KUKA KRL program: MyProgram_243().src

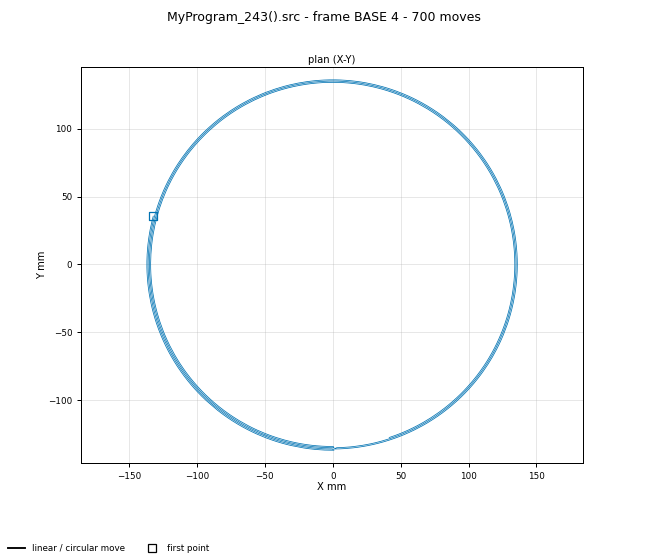
[picture p0: tool path of MyProgram_243().src in frame BASE 4, 700 of 700 moves have a stored position in this frame; points joined in program order, loops and branches not executed]
&ACCESS RVP
&REL 1
&PARAM TEMPLATE = C:\KRC\Roboter\Template\vorgabe
&PARAM EDITMASK = *
DEF MyProgram_243()
; ---- Setting reference (Base) ----
$BASE = BASE_DATA[4]

; --------------------------
; ---- Setting tool (TCP) ----
$TOOL = TOOL_DATA[3]
; --------------------------

$VEL.CP = VEL_APROX_PRINT
Startdeposition()
$VEL.CP = VEL_PRINT
LIN {X -132.1479,Y 35.5316,Z 162,A 162.612,B 22.5411,C -1.0275,E1 22.4083,E2 284.7882} C_DIS
LIN {X -132.9584,Y 32.3675,Z 162,A 163.9986,B 22.5412,C -1.024,E1 22.4074,E2 283.4017} C_DIS
LIN {X -133.7341,Y 28.9953,Z 162,A 165.3572,B 22.5416,C -1.0153,E1 22.4065,E2 282.0568} C_DIS
LIN {X -134.3965,Y 25.7509,Z 162,A 166.8499,B 22.5416,C -1.0157,E1 22.4057,E2 280.5534} C_DIS
LIN {X -134.985,Y 22.4628,Z 162,A 168.2719,B 22.5417,C -1.0122,E1 22.4051,E2 279.1309} C_DIS
LIN {X -135.5638,Y 18.6678,Z 162,A 170.017,B 22.5417,C -1.0132,E1 22.4044,E2 277.3716} C_DIS
LIN {X -136.0422,Y 14.7684,Z 162,A 171.5514,B 22.5421,C -1.0029,E1 22.4039,E2 275.8538} C_DIS
LIN {X -136.3695,Y 11.3551,Z 162,A 173.0277,B 22.5422,C -1.0001,E1 22.4035,E2 274.375} C_DIS
LIN {X -136.6388,Y 7.4678,Z 162,A 174.7811,B 22.5422,C -1.0003,E1 22.4032,E2 272.6092} C_DIS
LIN {X -136.821,Y 2.3704,Z 162,A 176.8126,B 22.5427,C -0.9887,E1 22.403,E2 270.5945} C_DIS
LIN {X -136.8263,Y -2.0499,Z 162,A 178.6813,B 22.5429,C -0.9835,E1 22.403,E2 268.7266} C_DIS
LIN {X -136.7134,Y -5.9516,Z 162,A -179.5726,B 22.5429,C -0.9833,E1 22.4033,E2 266.9694} C_DIS
LIN {X -136.4577,Y -10.2442,Z 162,A -177.8134,B 22.5432,C -0.9757,E1 22.4036,E2 265.2183} C_DIS
LIN {X -136.0949,Y -14.2787,Z 162,A -176.2336,B 22.5437,C -0.965,E1 22.404,E2 263.656} C_DIS
LIN {X -135.6787,Y -17.8001,Z 162,A -174.6843,B 22.5437,C -0.9632,E1 22.4045,E2 262.1009} C_DIS
LIN {X -135.101,Y -21.7679,Z 162,A -172.859,B 22.5437,C -0.9645,E1 22.4053,E2 260.2601} C_DIS
LIN {X -134.448,Y -25.4817,Z 162,A -171.4171,B 22.5442,C -0.9533,E1 22.406,E2 258.8378} C_DIS
LIN {X -133.8444,Y -28.4841,Z 162,A -170.0113,B 22.5441,C -0.9549,E1 22.4069,E2 257.4185} C_DIS
LIN {X -133.0086,Y -32.1595,Z 162,A -168.5445,B 22.5445,C -0.945,E1 22.4078,E2 255.9682} C_DIS
LIN {X -132.1539,Y -35.5092,Z 162,A -166.498,B 22.5436,C -0.9678,E1 22.4093,E2 253.8483} C_DIS
LIN {X -130.8595,Y -40.0158,Z 162,A -165.0549,B 22.5448,C -0.9381,E1 22.4104,E2 252.474} C_DIS
LIN {X -129.8351,Y -43.2241,Z 162,A -163.6072,B 22.5448,C -0.9356,E1 22.4117,E2 251.0236} C_DIS
LIN {X -128.378,Y -47.3813,Z 162,A -161.5655,B 22.5448,C -0.939,E1 22.4136,E2 248.9597} C_DIS
LIN {X -126.4379,Y -52.3363,Z 162,A -159.5206,B 22.5453,C -0.9242,E1 22.4157,E2 246.9411} C_DIS
LIN {X -125.0704,Y -55.5246,Z 162,A -157.4706,B 22.5444,C -0.9474,E1 22.4182,E2 244.8173} C_DIS
LIN {X -122.9248,Y -60.126,Z 162,A -155.4739,B 22.5449,C -0.9355,E1 22.4206,E2 242.8399} C_DIS
LIN {X -120.9842,Y -63.9405,Z 162,A -154.3142,B 22.5462,C -0.9014,E1 22.422,E2 241.7626} C_DIS
LIN {X -118.9843,Y -67.5927,Z 162,A -152.2799,B 22.5458,C -0.91,E1 22.4248,E2 239.6938} C_DIS
LIN {X -116.5755,Y -71.6669,Z 162,A -150.3113,B 22.5461,C -0.9041,E1 22.4276,E2 237.7294} C_DIS
LIN {X -114.3025,Y -75.2391,Z 162,A -148.0549,B 22.5454,C -0.9219,E1 22.4312,E2 235.4136} C_DIS
LIN {X -111.6085,Y -79.1811,Z 162,A -146.4975,B 22.5464,C -0.8963,E1 22.4336,E2 233.9147} C_DIS
LIN {X -109.6366,Y -81.8891,Z 162,A -145.0699,B 22.5464,C -0.894,E1 22.4359,E2 232.4854} C_DIS
LIN {X -106.8318,Y -85.5165,Z 162,A -143.1704,B 22.5467,C -0.8884,E1 22.4392,E2 230.5905} C_DIS
LIN {X -104.4579,Y -88.4003,Z 162,A -141.3214,B 22.5463,C -0.898,E1 22.4426,E2 228.7069} C_DIS
LIN {X -102.0287,Y -91.1928,Z 162,A -140.3003,B 22.5473,C -0.8699,E1 22.4444,E2 227.7543} C_DIS
LIN {X -99.6826,Y -93.7518,Z 162,A -138.5586,B 22.547,C -0.88,E1 22.4477,E2 225.9775} C_DIS
LIN {X -96.344,Y -97.1794,Z 162,A -136.6172,B 22.5472,C -0.8728,E1 22.4515,E2 224.0457} C_DIS
LIN {X -93.0775,Y -100.3126,Z 162,A -134.6531,B 22.5472,C -0.8721,E1 22.4555,E2 222.0744} C_DIS
LIN {X -84.7797,Y -107.4174,Z 162,A -130.3287,B 22.548,C -0.8514,E1 22.4647,E2 217.7853} C_DIS
LIN {X -80.9765,Y -110.3122,Z 162,A -128.1214,B 22.5478,C -0.8575,E1 22.4697,E2 215.5533} C_DIS
LIN {X -77.7183,Y -112.632,Z 162,A -126.346,B 22.5478,C -0.8594,E1 22.4737,E2 213.766} C_DIS
LIN {X -73.8799,Y -115.1857,Z 162,A -124.4429,B 22.5478,C -0.8551,E1 22.4782,E2 211.8674} C_DIS
LIN {X -69.9948,Y -117.587,Z 162,A -122.5683,B 22.5481,C -0.8504,E1 22.4826,E2 209.9985} C_DIS
LIN {X -66.2461,Y -119.739,Z 162,A -120.7348,B 22.5481,C -0.849,E1 22.4871,E2 208.1627} C_DIS
LIN {X -62.7854,Y -121.5897,Z 162,A -119.0231,B 22.5481,C -0.8501,E1 22.4914,E2 206.4428} C_DIS
LIN {X -59.1797,Y -123.3825,Z 162,A -117.3145,B 22.5481,C -0.8491,E1 22.4957,E2 204.7317} C_DIS
LIN {X -55.5104,Y -125.0767,Z 162,A -115.3139,B 22.5476,C -0.862,E1 22.5009,E2 202.692} C_DIS
LIN {X -51.6723,Y -126.7112,Z 162,A -113.931,B 22.5483,C -0.8427,E1 22.5043,E2 201.3562} C_DIS
LIN {X -48.8745,Y -127.8175,Z 162,A -112.5832,B 22.5483,C -0.8457,E1 22.5079,E2 199.9973} C_DIS
LIN {X -44.8525,Y -129.2816,Z 162,A -110.9547,B 22.5486,C -0.8362,E1 22.5121,E2 198.3899} C_DIS
LIN {X -41.5447,Y -130.3822,Z 162,A -109.4829,B 22.5486,C -0.8356,E1 22.516,E2 196.9167} C_DIS
LIN {X -37.9958,Y -131.4611,Z 162,A -107.8588,B 22.5485,C -0.838,E1 22.5204,E2 195.2835} C_DIS
LIN {X -33.7722,Y -132.6083,Z 162,A -106.1156,B 22.5487,C -0.8325,E1 22.525,E2 193.5517} C_DIS
LIN {X -30.5556,Y -133.3862,Z 162,A -104.7545,B 22.5487,C -0.8306,E1 22.5287,E2 192.1935} C_DIS
LIN {X -21.194,Y -135.1903,Z 162,A -100.7042,B 22.5487,C -0.8317,E1 22.5399,E2 188.1354} C_DIS
LIN {X -17.7477,Y -135.6855,Z 162,A -98.5879,B 22.5476,C -0.8638,E1 22.546,E2 185.9337} C_DIS
LIN {X -12.3536,Y -136.2845,Z 162,A -96.7009,B 22.5483,C -0.8445,E1 22.5511,E2 184.096} C_DIS
LIN {X -9.1175,Y -136.5392,Z 162,A -95.3192,B 22.5483,C -0.8456,E1 22.5549,E2 182.7108} C_DIS
LIN {X -5.827,Y -136.7182,Z 162,A -94.3815,B 22.549,C -0.8239,E1 22.5574,E2 181.8294} C_DIS
LIN {X 0.956,Y -136.8378,Z 162,A -91.1377,B 22.5483,C -0.8443,E1 22.5666,E2 178.5323} C_DIS
Enddeposition()
LIN {X 0.956,Y -136.8378,Z 162,A -91.1377,B 22.5483,C -0.8443,E1 22.5666,E2 178.5323} C_DIS
Startdeposition()
$VEL.CP = VEL_PRINT
LIN {X -0.2334,Y -135.9196,Z 162,A -92.5282,B 21.3065,C -0.6019,E1 21.3126,E2 180.4426} C_DIS
LIN {X -3.8269,Y -135.8649,Z 162,A -93.5596,B 21.3059,C -0.6237,E1 21.3099,E2 181.4142} C_DIS
LIN {X -7.1029,Y -135.7333,Z 162,A -95.1398,B 21.3062,C -0.6146,E1 21.3054,E2 183.0199} C_DIS
LIN {X -13.5908,Y -135.2388,Z 162,A -98.0002,B 21.3063,C -0.6094,E1 21.2974,E2 185.896} C_DIS
LIN {X -17.7059,Y -134.7604,Z 162,A -99.5578,B 21.3061,C -0.6183,E1 21.2932,E2 187.4305} C_DIS
LIN {X -21.7349,Y -134.171,Z 162,A -101.4303,B 21.3062,C -0.6118,E1 21.2879,E2 189.3229} C_DIS
LIN {X -28.2019,Y -132.9613,Z 162,A -103.9064,B 21.3058,C -0.6262,E1 21.2813,E2 191.7624} C_DIS
LIN {X -32.3871,Y -132.0045,Z 162,A -105.8123,B 21.3059,C -0.6229,E1 21.276,E2 193.6806} C_DIS
LIN {X -35.1696,Y -131.2895,Z 162,A -107.0688,B 21.3059,C -0.6216,E1 21.2726,E2 194.9428} C_DIS
LIN {X -38.4295,Y -130.3727,Z 162,A -108.5181,B 21.3059,C -0.6216,E1 21.2687,E2 196.3948} C_DIS
LIN {X -42.4293,Y -129.1272,Z 162,A -110.4038,B 21.3061,C -0.6177,E1 21.2637,E2 198.2954} C_DIS
LIN {X -46.4957,Y -127.7188,Z 162,A -112.3466,B 21.3061,C -0.6136,E1 21.2585,E2 200.2541} C_DIS
LIN {X -55.1136,Y -124.2434,Z 162,A -116.0722,B 21.3058,C -0.6261,E1 21.249,E2 203.9553} C_DIS
LIN {X -58.8057,Y -122.5386,Z 162,A -117.7449,B 21.3058,C -0.6299,E1 21.2448,E2 205.6224} C_DIS
LIN {X -62.2944,Y -120.8042,Z 162,A -119.3789,B 21.3057,C -0.6324,E1 21.2407,E2 207.2549} C_DIS
LIN {X -65.536,Y -119.0775,Z 162,A -121.0522,B 21.3057,C -0.629,E1 21.2365,E2 208.9432} C_DIS
LIN {X -69.4336,Y -116.8473,Z 162,A -122.9199,B 21.3057,C -0.6328,E1 21.232,E2 210.807} C_DIS
LIN {X -73.1219,Y -114.5753,Z 162,A -124.7704,B 21.3057,C -0.6345,E1 21.2277,E2 212.6598} C_DIS
LIN {X -76.9602,Y -112.0331,Z 162,A -126.6969,B 21.3055,C -0.6383,E1 21.2232,E2 214.5835} C_DIS
LIN {X -80.6257,Y -109.4249,Z 162,A -128.6706,B 21.3055,C -0.6382,E1 21.2187,E2 216.5658} C_DIS
LIN {X -83.2917,Y -107.4094,Z 162,A -130.0276,B 21.3054,C -0.6429,E1 21.2157,E2 217.9155} C_DIS
LIN {X -86.9347,Y -104.4832,Z 162,A -132.4983,B 21.3059,C -0.6251,E1 21.2103,E2 220.4466} C_DIS
LIN {X -90.5729,Y -101.3452,Z 162,A -134.0516,B 21.3052,C -0.6493,E1 21.2072,E2 221.9404} C_DIS
LIN {X -93.8703,Y -98.2987,Z 162,A -135.85,B 21.305,C -0.6572,E1 21.2035,E2 223.7257} C_DIS
LIN {X -96.946,Y -95.2668,Z 162,A -137.5121,B 21.3046,C -0.6679,E1 21.2003,E2 225.3667} C_DIS
LIN {X -99.0485,Y -93.0793,Z 162,A -139.0778,B 21.3049,C -0.6584,E1 21.1972,E2 226.9669} C_DIS
LIN {X -102.0742,Y -89.7511,Z 162,A -141.0897,B 21.3049,C -0.6577,E1 21.1934,E2 228.9914} C_DIS
LIN {X -105.3855,Y -85.8384,Z 162,A -143.1221,B 21.3046,C -0.6682,E1 21.1898,E2 231.0058} C_DIS
LIN {X -108.1096,Y -82.3812,Z 162,A -144.9286,B 21.3044,C -0.6748,E1 21.1867,E2 232.8045} C_DIS
LIN {X -110.4942,Y -79.1539,Z 162,A -146.6977,B 21.3044,C -0.6756,E1 21.1838,E2 234.5814} C_DIS
LIN {X -113.3531,Y -75.0031,Z 162,A -148.6448,B 21.304,C -0.6885,E1 21.1808,E2 236.5044} C_DIS
LIN {X -115.2076,Y -72.1223,Z 162,A -150.3202,B 21.3042,C -0.6825,E1 21.1783,E2 238.2067} C_DIS
LIN {X -117.4639,Y -68.3859,Z 162,A -152.1255,B 21.304,C -0.6888,E1 21.1757,E2 240.0056} C_DIS
LIN {X -119.6677,Y -64.4511,Z 162,A -154.0117,B 21.3038,C -0.6946,E1 21.1732,E2 241.8877} C_DIS
LIN {X -121.1916,Y -61.5335,Z 162,A -155.3534,B 21.3036,C -0.7004,E1 21.1714,E2 243.2219} C_DIS
LIN {X -124.3228,Y -54.9361,Z 162,A -158.4447,B 21.3034,C -0.7085,E1 21.1678,E2 246.311} C_DIS
LIN {X -125.5052,Y -52.1752,Z 162,A -159.7449,B 21.3034,C -0.7107,E1 21.1664,E2 247.6137} C_DIS
LIN {X -126.8199,Y -48.894,Z 162,A -161.2631,B 21.3032,C -0.7138,E1 21.1648,E2 249.1334} C_DIS
LIN {X -128.294,Y -44.8841,Z 162,A -163.1444,B 21.3032,C -0.7158,E1 21.163,E2 251.0221} C_DIS
LIN {X -129.5273,Y -41.1886,Z 162,A -164.7044,B 21.3029,C -0.7241,E1 21.1617,E2 252.5696} C_DIS
LIN {X -130.563,Y -37.7794,Z 162,A -166.5203,B 21.3032,C -0.7155,E1 21.1602,E2 254.4219} C_DIS
LIN {X -131.434,Y -34.6278,Z 162,A -167.5885,B 21.3026,C -0.7326,E1 21.1595,E2 255.4501} C_DIS
LIN {X -132.3079,Y -31.1286,Z 162,A -169.276,B 21.3026,C -0.7303,E1 21.1584,E2 257.1559} C_DIS
LIN {X -133.2279,Y -26.9106,Z 162,A -170.9656,B 21.3023,C -0.7413,E1 21.1574,E2 258.8268} C_DIS
LIN {X -133.7716,Y -24.0628,Z 162,A -172.2202,B 21.3023,C -0.7438,E1 21.1568,E2 260.0835} C_DIS
LIN {X -134.3449,Y -20.6232,Z 162,A -173.671,B 21.3021,C -0.7492,E1 21.1561,E2 261.5297} C_DIS
LIN {X -134.8662,Y -16.8982,Z 162,A -175.2631,B 21.3019,C -0.7538,E1 21.1556,E2 263.1203} C_DIS
LIN {X -135.1826,Y -14.132,Z 162,A -176.5632,B 21.3019,C -0.7523,E1 21.1552,E2 264.4339} C_DIS
LIN {X -135.5553,Y -9.9317,Z 162,A -178.2889,B 21.3017,C -0.7601,E1 21.1548,E2 266.1503} C_DIS
LIN {X -135.793,Y -5.8728,Z 162,A 179.9148,B 21.3017,C -0.7621,E1 21.1545,E2 267.9541} C_DIS
LIN {X -135.9038,Y -2.0291,Z 162,A 178.401,B 21.3013,C -0.7717,E1 21.1545,E2 269.4521} C_DIS
LIN {X -135.901,Y 2.1995,Z 162,A 176.5657,B 21.3012,C -0.7752,E1 21.1545,E2 271.2909} C_DIS
LIN {X -135.7975,Y 5.7565,Z 162,A 175.1116,B 21.3009,C -0.7819,E1 21.1545,E2 272.7369} C_DIS
LIN {X -135.6057,Y 9.2415,Z 162,A 173.5075,B 21.3009,C -0.7811,E1 21.1549,E2 274.3548} C_DIS
LIN {X -135.2923,Y 13.033,Z 162,A 171.9109,B 21.3008,C -0.7866,E1 21.1553,E2 275.9478} C_DIS
LIN {X -134.7943,Y 17.4468,Z 162,A 170.0685,B 21.3005,C -0.7938,E1 21.1559,E2 277.7834} C_DIS
LIN {X -134.3075,Y 20.8651,Z 162,A 168.6193,B 21.3003,C -0.7987,E1 21.1565,E2 279.2293} C_DIS
LIN {X -133.7052,Y 24.4337,Z 162,A 167.0858,B 21.3002,C -0.8032,E1 21.1572,E2 280.7613} C_DIS
LIN {X -132.9189,Y 28.3983,Z 162,A 165.3214,B 21.3001,C -0.8061,E1 21.1582,E2 282.5301} C_DIS
LIN {X -132.1192,Y 31.9113,Z 162,A 163.8484,B 21.2998,C -0.8127,E1 21.1591,E2 283.995} C_DIS
LIN {X -131.2604,Y 35.2787,Z 162,A 162.3572,B 21.2998,C -0.8162,E1 21.1602,E2 285.4869} C_DIS
LIN {X -130.2348,Y 38.9002,Z 162,A 160.7651,B 21.2995,C -0.8209,E1 21.1614,E2 287.077} C_DIS
LIN {X -129.1239,Y 42.4391,Z 162,A 159.126,B 21.2995,C -0.8226,E1 21.1628,E2 288.7226} C_DIS
LIN {X -127.8789,Y 46.0518,Z 162,A 157.5218,B 21.2993,C -0.8279,E1 21.1643,E2 290.3232} C_DIS
LIN {X -126.4348,Y 49.8846,Z 162,A 155.8123,B 21.2991,C -0.8338,E1 21.166,E2 292.0278} C_DIS
LIN {X -124.6618,Y 54.1596,Z 162,A 153.8509,B 21.2989,C -0.8392,E1 21.1681,E2 293.9871} C_DIS
LIN {X -123.2442,Y 57.3124,Z 162,A 152.347,B 21.2988,C -0.8416,E1 21.1699,E2 295.4942} C_DIS
LIN {X -121.3485,Y 61.2251,Z 162,A 150.6714,B 21.2983,C -0.8536,E1 21.1719,E2 297.1476} C_DIS
LIN {X -118.0764,Y 67.322,Z 162,A 147.6014,B 21.2983,C -0.8555,E1 21.176,E2 300.2315} C_DIS
LIN {X -116.2087,Y 70.4973,Z 162,A 145.9945,B 21.2982,C -0.8577,E1 21.1783,E2 301.8424} C_DIS
LIN {X -114.0464,Y 73.9439,Z 162,A 144.2065,B 21.2981,C -0.8594,E1 21.181,E2 303.6364} C_DIS
LIN {X -110.7896,Y 78.7407,Z 162,A 141.8266,B 21.2977,C -0.8687,E1 21.1848,E2 306.0046} C_DIS
LIN {X -106.8612,Y 83.9939,Z 162,A 139.0312,B 21.2975,C -0.8748,E1 21.1895,E2 308.7992} C_DIS
LIN {X -102.9226,Y 88.7763,Z 162,A 136.4415,B 21.2972,C -0.8823,E1 21.1941,E2 311.3822} C_DIS
LIN {X -100.3087,Y 91.7201,Z 162,A 134.6734,B 21.2972,C -0.8819,E1 21.1974,E2 313.1609} C_DIS
LIN {X -97.2658,Y 94.9407,Z 162,A 132.7521,B 21.2972,C -0.8842,E1 21.2012,E2 315.0859} C_DIS
LIN {X -94.0928,Y 98.0861,Z 162,A 130.8858,B 21.2969,C -0.8893,E1 21.2049,E2 316.9473} C_DIS
LIN {X -90.9182,Y 101.0359,Z 162,A 129.0267,B 21.2969,C -0.8921,E1 21.2087,E2 318.8076} C_DIS
LIN {X -87.6094,Y 103.9181,Z 162,A 127.2544,B 21.2965,C -0.8994,E1 21.2124,E2 320.5679} C_DIS
LIN {X -84.4386,Y 106.5104,Z 162,A 125.3203,B 21.2967,C -0.8943,E1 21.2167,E2 322.5247} C_DIS
LIN {X -80.6388,Y 109.4153,Z 162,A 123.3832,B 21.2964,C -0.9018,E1 21.221,E2 324.4495} C_DIS
LIN {X -75.1849,Y 113.2326,Z 162,A 120.4463,B 21.2964,C -0.9017,E1 21.2278,E2 327.3985} C_DIS
LIN {X -70.65,Y 116.1163,Z 162,A 118.3043,B 21.296,C -0.9111,E1 21.2328,E2 329.5226} C_DIS
LIN {X -66.7886,Y 118.3792,Z 162,A 116.2717,B 21.2962,C -0.9081,E1 21.2378,E2 331.5706} C_DIS
LIN {X -61.6496,Y 121.1324,Z 162,A 113.9949,B 21.2957,C -0.9199,E1 21.2434,E2 333.8224} C_DIS
LIN {X -58.3357,Y 122.7631,Z 162,A 112.49,B 21.2955,C -0.9245,E1 21.2471,E2 335.3192} C_DIS
LIN {X -54.6496,Y 124.4499,Z 162,A 110.8257,B 21.2953,C -0.9289,E1 21.2513,E2 336.9762} C_DIS
LIN {X -52.2373,Y 125.4793,Z 162,A 109.3523,B 21.2959,C -0.9146,E1 21.2553,E2 338.493} C_DIS
LIN {X -48.9956,Y 126.7804,Z 162,A 108.2083,B 21.2952,C -0.9306,E1 21.2581,E2 339.5956} C_DIS
LIN {X -45.4252,Y 128.1048,Z 162,A 106.6215,B 21.2952,C -0.9334,E1 21.2623,E2 341.1786} C_DIS
LIN {X -42.5094,Y 129.1005,Z 162,A 105.3219,B 21.2951,C -0.9349,E1 21.2657,E2 342.477} C_DIS
LIN {X -35.9614,Y 131.0764,Z 162,A 102.4892,B 21.2948,C -0.9401,E1 21.2733,E2 345.3009} C_DIS
LIN {X -31.8419,Y 132.1359,Z 162,A 100.5975,B 21.2949,C -0.9375,E1 21.2784,E2 347.2031} C_DIS
LIN {X -28.6415,Y 132.8664,Z 162,A 99.2454,B 21.2949,C -0.9401,E1 21.2821,E2 348.5501} C_DIS
LIN {X -25.4806,Y 133.5087,Z 162,A 97.8355,B 21.2949,C -0.9389,E1 21.286,E2 349.965} C_DIS
LIN {X -22.2396,Y 134.0868,Z 162,A 96.4615,B 21.2949,C -0.9405,E1 21.2897,E2 351.3363} C_DIS
LIN {X -18.9892,Y 134.5857,Z 162,A 95.0405,B 21.2949,C -0.9398,E1 21.2937,E2 352.7606} C_DIS
LIN {X -13.679,Y 135.2303,Z 162,A 92.7643,B 21.2949,C -0.94,E1 21.3,E2 355.0379} C_DIS
LIN {X -9.9539,Y 135.5537,Z 162,A 91.1718,B 21.2949,C -0.94,E1 21.3044,E2 356.6313} C_DIS
LIN {X -6.3293,Y 135.7721,Z 162,A 89.7311,B 21.2947,C -0.9445,E1 21.3084,E2 358.0602} C_DIS
LIN {X -2.3794,Y 135.898,Z 162,A 87.9675,B 21.2948,C -0.9405,E1 21.3134,E2 359.8348} C_DIS
LIN {X 2.0503,Y 135.9034,Z 162,A 86.1664,B 21.2947,C -0.9437,E1 21.3184,E2 361.6269} C_DIS
LIN {X 5.7146,Y 135.7992,Z 162,A 84.657,B 21.2947,C -0.9454,E1 21.3226,E2 363.1313} C_DIS
LIN {X 10.3482,Y 135.5249,Z 162,A 82.6398,B 21.2947,C -0.9426,E1 21.3282,E2 365.1551} C_DIS
LIN {X 13.4186,Y 135.2553,Z 162,A 81.287,B 21.2948,C -0.94,E1 21.332,E2 366.514} C_DIS
LIN {X 17.5932,Y 134.7751,Z 162,A 79.5677,B 21.2948,C -0.942,E1 21.3367,E2 368.2264} C_DIS
LIN {X 20.864,Y 134.3076,Z 162,A 77.8795,B 21.2953,C -0.9283,E1 21.3415,E2 369.9504} C_DIS
LIN {X 24.3503,Y 133.7201,Z 162,A 76.7633,B 21.2947,C -0.9445,E1 21.3444,E2 371.0206} C_DIS
LIN {X 27.8278,Y 133.0413,Z 162,A 75.2567,B 21.2947,C -0.9432,E1 21.3486,E2 372.5286} C_DIS
LIN {X 30.5921,Y 132.4313,Z 162,A 74.0865,B 21.2947,C -0.9436,E1 21.3517,E2 373.6958} C_DIS
LIN {X 33.5926,Y 131.7018,Z 162,A 72.7585,B 21.2947,C -0.9416,E1 21.3554,E2 375.0269} C_DIS
LIN {X 36.7603,Y 130.853,Z 162,A 71.3771,B 21.2948,C -0.9407,E1 21.3591,E2 376.4081} C_DIS
LIN {X 39.9209,Y 129.9236,Z 162,A 69.916,B 21.295,C -0.9363,E1 21.363,E2 377.8781} C_DIS
LIN {X 43.3175,Y 128.8314,Z 162,A 68.1588,B 21.2955,C -0.9235,E1 21.3677,E2 379.6664} C_DIS
LIN {X 46.5345,Y 127.7049,Z 162,A 66.244,B 21.2965,C -0.9005,E1 21.3729,E2 381.6395} C_DIS
LIN {X 52.0712,Y 125.5486,Z 162,A 64.7367,B 21.2947,C -0.9433,E1 21.3765,E2 383.0252} C_DIS
LIN {X 55.7247,Y 123.97,Z 162,A 62.8499,B 21.2952,C -0.9318,E1 21.3814,E2 384.9382} C_DIS
LIN {X 59.0495,Y 122.422,Z 162,A 61.3314,B 21.2952,C -0.9312,E1 21.3852,E2 386.4537} C_DIS
LIN {X 61.9759,Y 120.9663,Z 162,A 59.9154,B 21.2954,C -0.9276,E1 21.3888,E2 387.8748} C_DIS
LIN {X 65.6585,Y 119.0097,Z 162,A 58.0907,B 21.2956,C -0.9221,E1 21.3933,E2 389.7083} C_DIS
LIN {X 69.5194,Y 116.7962,Z 162,A 56.2584,B 21.2956,C -0.9214,E1 21.3977,E2 391.536} C_DIS
LIN {X 73.2636,Y 114.4846,Z 162,A 54.3926,B 21.2958,C -0.918,E1 21.4021,E2 393.404} C_DIS
LIN {X 77.0918,Y 111.9428,Z 162,A 52.4689,B 21.2958,C -0.9154,E1 21.4065,E2 395.3271} C_DIS
LIN {X 81.2712,Y 108.9463,Z 162,A 50.5979,B 21.2954,C -0.9255,E1 21.4107,E2 397.1625} C_DIS
LIN {X 88.4978,Y 103.1625,Z 162,A 46.7313,B 21.2957,C -0.9197,E1 21.4192,E2 401.0275} C_DIS
LIN {X 91.8269,Y 100.2105,Z 162,A 44.5748,B 21.2964,C -0.9027,E1 21.4237,E2 403.2202} C_DIS
LIN {X 94.9661,Y 97.2409,Z 162,A 42.9591,B 21.2961,C -0.9086,E1 21.4269,E2 404.8118} C_DIS
LIN {X 97.176,Y 95.0323,Z 162,A 41.4452,B 21.2966,C -0.8965,E1 21.4299,E2 406.3512} C_DIS
LIN {X 100.1432,Y 91.9002,Z 162,A 39.5007,B 21.297,C -0.8865,E1 21.4336,E2 408.3129} C_DIS
LIN {X 103.4604,Y 88.1491,Z 162,A 37.5101,B 21.297,C -0.8874,E1 21.4373,E2 410.2904} C_DIS
LIN {X 106.4331,Y 84.5358,Z 162,A 35.4801,B 21.2973,C -0.8799,E1 21.4408,E2 412.3296} C_DIS
LIN {X 108.7196,Y 81.5749,Z 162,A 33.3572,B 21.2984,C -0.8503,E1 21.4445,E2 414.5214} C_DIS
LIN {X 111.9869,Y 77.0275,Z 162,A 31.9068,B 21.297,C -0.8874,E1 21.4467,E2 415.8617} C_DIS
LIN {X 113.7639,Y 74.379,Z 162,A 30.2771,B 21.2977,C -0.8703,E1 21.4492,E2 417.5285} C_DIS
LIN {X 116.1563,Y 70.5839,Z 162,A 28.4077,B 21.2978,C -0.8664,E1 21.452,E2 419.3973} C_DIS
LIN {X 118.3523,Y 66.8363,Z 162,A 26.5908,B 21.298,C -0.8622,E1 21.4545,E2 421.2146} C_DIS
LIN {X 120.461,Y 62.9519,Z 162,A 24.8895,B 21.2979,C -0.8649,E1 21.4567,E2 422.8978} C_DIS
LIN {X 122.1881,Y 59.5336,Z 162,A 23.2546,B 21.2981,C -0.8594,E1 21.4588,E2 424.5374} C_DIS
LIN {X 123.4847,Y 56.7923,Z 162,A 21.9888,B 21.2982,C -0.8564,E1 21.4603,E2 425.8032} C_DIS
LIN {X 124.8021,Y 53.8349,Z 162,A 20.5998,B 21.2984,C -0.8513,E1 21.4618,E2 427.197} C_DIS
LIN {X 126.3015,Y 50.2205,Z 162,A 18.7033,B 21.299,C -0.8346,E1 21.4638,E2 429.1266} C_DIS
LIN {X 129.0338,Y 42.7098,Z 162,A 15.0167,B 21.3,C -0.8095,E1 21.4672,E2 432.8571} C_DIS
LIN {X 130.5435,Y 37.846,Z 162,A 13.5687,B 21.299,C -0.8366,E1 21.4683,E2 434.2212} C_DIS
LIN {X 131.3307,Y 35.015,Z 162,A 12.2659,B 21.2992,C -0.8297,E1 21.4693,E2 435.5339} C_DIS
LIN {X 132.1821,Y 31.6503,Z 162,A 10.8073,B 21.2994,C -0.8255,E1 21.4703,E2 436.9941} C_DIS
LIN {X 132.9609,Y 28.2037,Z 162,A 9.4265,B 21.2994,C -0.8261,E1 21.4711,E2 438.3635} C_DIS
LIN {X 133.5085,Y 25.4818,Z 162,A 8.165,B 21.2996,C -0.8181,E1 21.4718,E2 439.6381} C_DIS
LIN {X 134.2214,Y 21.4212,Z 162,A 6.2718,B 21.3001,C -0.8051,E1 21.4727,E2 441.5535} C_DIS
LIN {X 134.8708,Y 16.8617,Z 162,A 4.4116,B 21.3001,C -0.8029,E1 21.4733,E2 443.4066} C_DIS
LIN {X 135.3133,Y 12.8141,Z 162,A 2.7455,B 21.3003,C -0.8,E1 21.4738,E2 445.069} C_DIS
LIN {X 135.6885,Y 7.919,Z 162,A 0.677,B 21.3005,C -0.7934,E1 21.4742,E2 447.1407} C_DIS
LIN {X 135.8661,Y 3.7808,Z 162,A -0.9786,B 21.3005,C -0.7923,E1 21.4744,E2 448.7878} C_DIS
LIN {X 135.9212,Y -0.1669,Z 162,A -2.79,B 21.301,C -0.7798,E1 21.4744,E2 450.6205} C_DIS
LIN {X 135.8354,Y -4.7856,Z 162,A -4.5729,B 21.301,C -0.7815,E1 21.4743,E2 452.3859} C_DIS
LIN {X 135.6696,Y -8.2265,Z 162,A -5.988,B 21.301,C -0.7787,E1 21.4741,E2 453.7987} C_DIS
LIN {X 135.3816,Y -12.0885,Z 162,A -7.6074,B 21.3012,C -0.7741,E1 21.4737,E2 455.4193} C_DIS
LIN {X 135.0135,Y -15.6655,Z 162,A -9.3366,B 21.3017,C -0.7589,E1 21.4731,E2 457.1778} C_DIS
LIN {X 134.2632,Y -21.151,Z 162,A -11.4057,B 21.3015,C -0.7643,E1 21.4723,E2 459.2176} C_DIS
LIN {X 133.7707,Y -24.0677,Z 162,A -12.6976,B 21.3018,C -0.7581,E1 21.4717,E2 460.5172} C_DIS
LIN {X 133.0162,Y -27.9478,Z 162,A -14.4194,B 21.302,C -0.7501,E1 21.4707,E2 462.2489} C_DIS
LIN {X 131.8917,Y -32.8445,Z 162,A -16.3162,B 21.3019,C -0.7542,E1 21.4695,E2 464.1215} C_DIS
LIN {X 130.7338,Y -37.1864,Z 162,A -18.2734,B 21.3022,C -0.7452,E1 21.4681,E2 466.0898} C_DIS
LIN {X 129.6235,Y -40.8873,Z 162,A -20.2572,B 21.3029,C -0.7229,E1 21.4664,E2 468.121} C_DIS
LIN {X 128.5078,Y -44.2674,Z 162,A -21.1751,B 21.3021,C -0.7466,E1 21.4657,E2 468.9682} C_DIS
LIN {X 125.7263,Y -51.6457,Z 162,A -24.7839,B 21.3029,C -0.7224,E1 21.462,E2 472.6189} C_DIS
LIN {X 124.0015,Y -55.6545,Z 162,A -26.5262,B 21.3029,C -0.7217,E1 21.4601,E2 474.352} C_DIS
LIN {X 122.4879,Y -58.9117,Z 162,A -28.0176,B 21.3031,C -0.7183,E1 21.4583,E2 475.8431} C_DIS
LIN {X 120.6786,Y -62.5377,Z 162,A -29.8002,B 21.3033,C -0.7096,E1 21.456,E2 477.6381} C_DIS
LIN {X 117.5764,Y -68.1916,Z 162,A -32.284,B 21.3033,C -0.7131,E1 21.4527,E2 480.0968} C_DIS
LIN {X 114.3258,Y -73.5118,Z 162,A -35.0612,B 21.3037,C -0.6984,E1 21.4486,E2 482.8973} C_DIS
LIN {X 110.9812,Y -78.4697,Z 162,A -37.4222,B 21.3037,C -0.6992,E1 21.4449,E2 485.2422} C_DIS
LIN {X 108.885,Y -81.3535,Z 162,A -39.1174,B 21.3041,C -0.6859,E1 21.442,E2 486.9642} C_DIS
LIN {X 106.1867,Y -84.8453,Z 162,A -40.9316,B 21.3041,C -0.6832,E1 21.4389,E2 488.7756} C_DIS
LIN {X 103.4742,Y -88.1328,Z 162,A -42.7384,B 21.3043,C -0.6781,E1 21.4357,E2 490.5865} C_DIS
LIN {X 100.4722,Y -91.5407,Z 162,A -44.6313,B 21.3044,C -0.6743,E1 21.4321,E2 492.4797} C_DIS
LIN {X 97.5178,Y -94.6816,Z 162,A -46.4227,B 21.3045,C -0.6711,E1 21.4287,E2 494.2705} C_DIS
LIN {X 94.7258,Y -97.4749,Z 162,A -48.1433,B 21.3047,C -0.6645,E1 21.4253,E2 496.0007} C_DIS
LIN {X 91.3653,Y -100.6314,Z 162,A -50.0386,B 21.3048,C -0.6623,E1 21.4214,E2 497.8927} C_DIS
LIN {X 88.052,Y -103.5429,Z 162,A -51.8966,B 21.3049,C -0.6582,E1 21.4174,E2 499.7533} C_DIS
LIN {X 84.5904,Y -106.3896,Z 162,A -53.7678,B 21.305,C -0.6549,E1 21.4134,E2 501.625} C_DIS
LIN {X 80.9725,Y -109.1687,Z 162,A -55.6773,B 21.3051,C -0.6516,E1 21.4091,E2 503.5354} C_DIS
LIN {X 77.3228,Y -111.7837,Z 162,A -57.5893,B 21.3053,C -0.6468,E1 21.4048,E2 505.4524} C_DIS
LIN {X 73.6704,Y -114.224,Z 162,A -59.4343,B 21.3053,C -0.6436,E1 21.4004,E2 507.299} C_DIS
LIN {X 69.6042,Y -116.7456,Z 162,A -61.3715,B 21.3053,C -0.6436,E1 21.3958,E2 509.2288} C_DIS
LIN {X 65.7737,Y -118.9458,Z 162,A -63.4378,B 21.3057,C -0.6308,E1 21.3907,E2 511.323} C_DIS
LIN {X 60.0343,Y -121.9411,Z 162,A -65.9312,B 21.3055,C -0.6375,E1 21.3846,E2 513.79} C_DIS
LIN {X 56.4086,Y -123.6621,Z 162,A -67.7346,B 21.3057,C -0.6296,E1 21.38,E2 515.6094} C_DIS
LIN {X 51.8056,Y -125.6596,Z 162,A -69.7892,B 21.3057,C -0.6294,E1 21.3747,E2 517.6587} C_DIS
LIN {X 47.9137,Y -127.1932,Z 162,A -71.8054,B 21.3061,C -0.6153,E1 21.3694,E2 519.7085} C_DIS
LIN {X 44.5649,Y -128.4046,Z 162,A -72.9651,B 21.3058,C -0.6293,E1 21.3664,E2 520.8269} C_DIS
LIN {X 41.1726,Y -129.5324,Z 162,A -74.5035,B 21.3058,C -0.6261,E1 21.3623,E2 522.3707} C_DIS
LIN {X 36.936,Y -130.8039,Z 162,A -76.4062,B 21.306,C -0.6223,E1 21.3572,E2 524.2799} C_DIS
LIN {X 33.2447,Y -131.7901,Z 162,A -77.9143,B 21.3059,C -0.6254,E1 21.3532,E2 525.7766} C_DIS
LIN {X 30.0368,Y -132.5582,Z 162,A -79.2964,B 21.3059,C -0.6245,E1 21.3494,E2 527.1588} C_DIS
LIN {X 26.509,Y -133.3097,Z 162,A -80.8135,B 21.3059,C -0.6234,E1 21.3453,E2 528.6768} C_DIS
LIN {X 22.7358,Y -134.004,Z 162,A -82.4793,B 21.306,C -0.6199,E1 21.3407,E2 530.3499} C_DIS
LIN {X 18.458,Y -134.6614,Z 162,A -84.2298,B 21.306,C -0.6221,E1 21.3359,E2 532.0925} C_DIS
LIN {X 15.0722,Y -135.0814,Z 162,A -85.8831,B 21.3063,C -0.6114,E1 21.3312,E2 533.7739} C_DIS
LIN {X 9.132,Y -135.6137,Z 162,A -88.3368,B 21.3063,C -0.613,E1 21.3244,E2 536.2216} C_DIS
LIN {X 5.1747,Y -135.8202,Z 162,A -89.921,B 21.3061,C -0.6164,E1 21.32,E2 537.7959} C_DIS
LIN {X 0.9468,Y -135.9079,Z 162,A -91.1941,B 21.3055,C -0.6394,E1 21.3166,E2 539.0054} C_DIS
Enddeposition()
LIN {X 0.9468,Y -135.9079,Z 162,A -91.1941,B 21.3055,C -0.6394,E1 21.3166,E2 539.0054} C_DIS
Startdeposition()
$VEL.CP = VEL_PRINT
LIN {X 2.9964,Y -134.9648,Z 162,A -89.8352,B 20.1418,C -0.4915,E1 20.1525,E2 537.9529} C_DIS
LIN {X 6.3819,Y -134.8456,Z 162,A -88.3556,B 20.1418,C -0.4938,E1 20.1566,E2 536.4671} C_DIS
LIN {X 9.7799,Y -134.6412,Z 162,A -87.0405,B 20.1419,C -0.4888,E1 20.1603,E2 535.1674} C_DIS
LIN {X 12.4989,Y -134.4166,Z 162,A -85.931,B 20.1419,C -0.4872,E1 20.1633,E2 534.0633} C_DIS
LIN {X 15.216,Y -134.1378,Z 162,A -84.5171,B 20.1417,C -0.4989,E1 20.1673,E2 532.6166} C_DIS
LIN {X 18.6912,Y -133.6962,Z 162,A -83.1451,B 20.1417,C -0.4948,E1 20.1711,E2 531.258} C_DIS
LIN {X 21.907,Y -133.2067,Z 162,A -81.7452,B 20.1417,C -0.4966,E1 20.175,E2 529.8547} C_DIS
LIN {X 24.9399,Y -132.6726,Z 162,A -80.6014,B 20.1419,C -0.4904,E1 20.1781,E2 528.7303} C_DIS
LIN {X 27.7029,Y -132.1251,Z 162,A -79.1445,B 20.1416,C -0.5029,E1 20.1821,E2 527.2397} C_DIS
LIN {X 31.3327,Y -131.3095,Z 162,A -77.6527,B 20.1416,C -0.5005,E1 20.1862,E2 525.7575} C_DIS
LIN {X 35.5712,Y -130.2274,Z 162,A -75.7102,B 20.1415,C -0.5061,E1 20.1914,E2 523.8026} C_DIS
LIN {X 39.0964,Y -129.2109,Z 162,A -74.4231,B 20.1417,C -0.4958,E1 20.1948,E2 522.548} C_DIS
LIN {X 41.8652,Y -128.3425,Z 162,A -72.9154,B 20.1414,C -0.5095,E1 20.1989,E2 521.0044} C_DIS
LIN {X 45.0037,Y -127.2759,Z 162,A -71.5195,B 20.1414,C -0.5107,E1 20.2026,E2 519.6085} C_DIS
LIN {X 48.5056,Y -125.9809,Z 162,A -70.0594,B 20.1414,C -0.5072,E1 20.2064,E2 518.1624} C_DIS
LIN {X 51.6195,Y -124.7373,Z 162,A -68.6395,B 20.1414,C -0.5091,E1 20.21,E2 516.7414} C_DIS
LIN {X 54.7168,Y -123.41,Z 162,A -67.2204,B 20.1414,C -0.5106,E1 20.2137,E2 515.3222} C_DIS
LIN {X 57.4276,Y -122.1743,Z 162,A -65.8291,B 20.1412,C -0.5182,E1 20.2172,E2 513.9135} C_DIS
LIN {X 60.4848,Y -120.69,Z 162,A -64.5146,B 20.1412,C -0.5147,E1 20.2205,E2 512.6136} C_DIS
LIN {X 63.6963,Y -119.0258,Z 162,A -62.8729,B 20.1412,C -0.522,E1 20.2246,E2 510.9566} C_DIS
LIN {X 67.8288,Y -116.7202,Z 162,A -60.9061,B 20.1411,C -0.5236,E1 20.2294,E2 508.9926} C_DIS
LIN {X 71.5152,Y -114.4986,Z 162,A -59.0864,B 20.141,C -0.5266,E1 20.2337,E2 507.1715} C_DIS
LIN {X 74.7667,Y -112.4023,Z 162,A -57.5289,B 20.141,C -0.5259,E1 20.2373,E2 505.6226} C_DIS
LIN {X 78.0881,Y -110.1211,Z 162,A -55.7417,B 20.1408,C -0.5328,E1 20.2414,E2 503.8235} C_DIS
LIN {X 81.666,Y -107.4949,Z 162,A -53.9518,B 20.1408,C -0.5324,E1 20.2454,E2 502.0428} C_DIS
LIN {X 84.5732,Y -105.2223,Z 162,A -52.3936,B 20.1408,C -0.5353,E1 20.2488,E2 500.4836} C_DIS
LIN {X 87.609,Y -102.7084,Z 162,A -50.6513,B 20.1406,C -0.5421,E1 20.2526,E2 498.7302} C_DIS
LIN {X 90.9781,Y -99.7367,Z 162,A -48.7458,B 20.1405,C -0.5464,E1 20.2565,E2 496.822} C_DIS
LIN {X 94.2145,Y -96.6856,Z 162,A -46.957,B 20.1405,C -0.5462,E1 20.2601,E2 495.0431} C_DIS
LIN {X 96.6856,Y -94.2145,Z 162,A -45.4077,B 20.1403,C -0.5528,E1 20.2632,E2 493.4833} C_DIS
LIN {X 99.6826,Y -91.0377,Z 162,A -43.5616,B 20.1403,C -0.557,E1 20.2667,E2 491.6353} C_DIS
LIN {X 102.5732,Y -87.768,Z 162,A -41.8007,B 20.1402,C -0.5574,E1 20.2699,E2 489.8832} C_DIS
LIN {X 104.8062,Y -85.089,Z 162,A -40.2785,B 20.14,C -0.5631,E1 20.2726,E2 488.3534} C_DIS
LIN {X 107.4264,Y -81.7556,Z 162,A -38.4918,B 20.14,C -0.5673,E1 20.2757,E2 486.5656} C_DIS
LIN {X 109.7412,Y -78.6204,Z 162,A -36.8113,B 20.1398,C -0.5729,E1 20.2784,E2 484.8791} C_DIS
LIN {X 112.0368,Y -75.3142,Z 162,A -35.2061,B 20.1398,C -0.5728,E1 20.2809,E2 483.2844} C_DIS
LIN {X 114.0392,Y -72.2455,Z 162,A -33.6629,B 20.1397,C -0.5765,E1 20.2833,E2 481.7401} C_DIS
LIN {X 116.1234,Y -68.8459,Z 162,A -31.9712,B 20.1395,C -0.5812,E1 20.2857,E2 480.0458} C_DIS
LIN {X 117.9923,Y -65.5909,Z 162,A -30.2923,B 20.1393,C -0.5897,E1 20.288,E2 478.3534} C_DIS
LIN {X 120.1017,Y -61.6404,Z 162,A -28.634,B 20.1395,C -0.5841,E1 20.2902,E2 476.7227} C_DIS
LIN {X 121.6176,Y -58.5927,Z 162,A -27.086,B 20.1392,C -0.593,E1 20.2921,E2 475.1594} C_DIS
LIN {X 122.8858,Y -55.8887,Z 162,A -25.8293,B 20.1392,C -0.5962,E1 20.2936,E2 473.902} C_DIS
LIN {X 124.3602,Y -52.5224,Z 162,A -24.3953,B 20.1392,C -0.5951,E1 20.2951,E2 472.4812} C_DIS
LIN {X 125.5196,Y -49.6921,Z 162,A -22.9958,B 20.1389,C -0.6037,E1 20.2966,E2 471.0669} C_DIS
LIN {X 126.8464,Y -46.1948,Z 162,A -21.3812,B 20.1387,C -0.6097,E1 20.2982,E2 469.4462} C_DIS
LIN {X 127.9469,Y -43.0531,Z 162,A -20.0248,B 20.1387,C -0.6114,E1 20.2994,E2 468.0946} C_DIS
LIN {X 128.8446,Y -40.2932,Z 162,A -18.8018,B 20.1386,C -0.6148,E1 20.3004,E2 466.8708} C_DIS
LIN {X 129.8924,Y -36.769,Z 162,A -17.2565,B 20.1385,C -0.6189,E1 20.3016,E2 465.3248} C_DIS
LIN {X 130.743,Y -33.6196,Z 162,A -16.0294,B 20.1385,C -0.6159,E1 20.3025,E2 464.1152} C_DIS
LIN {X 131.4264,Y -30.8478,Z 162,A -14.5679,B 20.1381,C -0.6312,E1 20.3035,E2 462.6203} C_DIS
LIN {X 132.2015,Y -27.3272,Z 162,A -13.3119,B 20.1383,C -0.6234,E1 20.3042,E2 461.3963} C_DIS
LIN {X 132.7443,Y -24.5647,Z 162,A -11.9852,B 20.138,C -0.6332,E1 20.3049,E2 460.0511} C_DIS
LIN {X 133.3432,Y -21.0623,Z 162,A -10.6331,B 20.1381,C -0.6308,E1 20.3055,E2 458.7162} C_DIS
LIN {X 133.7494,Y -18.3186,Z 162,A -9.2137,B 20.1377,C -0.6457,E1 20.3061,E2 457.2643} C_DIS
LIN {X 134.1776,Y -14.8462,Z 162,A -7.9947,B 20.1379,C -0.6381,E1 20.3065,E2 456.0765} C_DIS
LIN {X 134.4791,Y -11.8097,Z 162,A -6.4867,B 20.1375,C -0.652,E1 20.3069,E2 454.5396} C_DIS
LIN {X 134.7346,Y -8.3961,Z 162,A -5.1187,B 20.1375,C -0.6527,E1 20.3071,E2 453.1799} C_DIS
LIN {X 134.878,Y -5.656,Z 162,A -3.9829,B 20.1374,C -0.655,E1 20.3073,E2 452.0459} C_DIS
LIN {X 134.9648,Y -2.9964,Z 162,A -2.864,B 20.1373,C -0.6581,E1 20.3073,E2 450.9266} C_DIS
LIN {X 134.9978,Y 0.3023,Z 162,A -1.3289,B 20.1369,C -0.6688,E1 20.3073,E2 449.3723} C_DIS
LIN {X 134.9307,Y 4.226,Z 162,A 0.3065,B 20.1369,C -0.6727,E1 20.3073,E2 447.7381} C_DIS
LIN {X 134.765,Y 7.9031,Z 162,A 1.5947,B 20.1371,C -0.6649,E1 20.3071,E2 446.4819} C_DIS
LIN {X 134.5507,Y 10.9618,Z 162,A 3.0253,B 20.1367,C -0.675,E1 20.3068,E2 445.033} C_DIS
LIN {X 134.2448,Y 14.2214,Z 162,A 4.4381,B 20.1366,C -0.6804,E1 20.3064,E2 443.6153} C_DIS
LIN {X 133.8528,Y 17.5297,Z 162,A 5.8378,B 20.1364,C -0.6841,E1 20.3059,E2 442.2153} C_DIS
LIN {X 133.3432,Y 21.0623,Z 162,A 7.4728,B 20.1361,C -0.6944,E1 20.3052,E2 440.5629} C_DIS
LIN {X 132.6726,Y 24.9399,Z 162,A 9.039,B 20.1361,C -0.6947,E1 20.3044,E2 439.0074} C_DIS
LIN {X 131.6997,Y 29.6511,Z 162,A 11.0056,B 20.1361,C -0.6975,E1 20.3033,E2 437.0473} C_DIS
LIN {X 130.9134,Y 32.9479,Z 162,A 12.4607,B 20.1358,C -0.7026,E1 20.3023,E2 435.588} C_DIS
LIN {X 130.0357,Y 36.2567,Z 162,A 13.7948,B 20.1358,C -0.7015,E1 20.3013,E2 434.2668} C_DIS
LIN {X 129.2109,Y 39.0964,Z 162,A 14.9782,B 20.1358,C -0.702,E1 20.3004,E2 433.0908} C_DIS
LIN {X 128.3425,Y 41.8652,Z 162,A 16.4701,B 20.1353,C -0.7176,E1 20.2991,E2 431.5647} C_DIS
LIN {X 127.2759,Y 45.0037,Z 162,A 17.8921,B 20.1352,C -0.7224,E1 20.2978,E2 430.1389} C_DIS
LIN {X 125.9809,Y 48.5056,Z 162,A 19.3229,B 20.1352,C -0.7199,E1 20.2964,E2 428.7253} C_DIS
LIN {X 124.7373,Y 51.6195,Z 162,A 20.7373,B 20.1352,C -0.7236,E1 20.2949,E2 427.3102} C_DIS
LIN {X 123.41,Y 54.7168,Z 162,A 22.1967,B 20.1349,C -0.729,E1 20.2933,E2 425.8453} C_DIS
LIN {X 122.1743,Y 57.4276,Z 162,A 23.5381,B 20.1347,C -0.736,E1 20.2917,E2 424.4928} C_DIS
LIN {X 120.69,Y 60.4848,Z 162,A 24.8485,B 20.1347,C -0.734,E1 20.2901,E2 423.1973} C_DIS
LIN {X 119.0258,Y 63.6963,Z 162,A 26.4858,B 20.1345,C -0.7428,E1 20.2879,E2 421.5454} C_DIS
LIN {X 116.7202,Y 67.8288,Z 162,A 28.4478,B 20.1343,C -0.7461,E1 20.2852,E2 419.587} C_DIS
LIN {X 114.4986,Y 71.5152,Z 162,A 30.2639,B 20.1342,C -0.7503,E1 20.2826,E2 417.7703} C_DIS
LIN {X 112.2632,Y 74.9752,Z 162,A 31.9845,B 20.1341,C -0.7535,E1 20.2799,E2 416.0513} C_DIS
LIN {X 110.0663,Y 78.1658,Z 162,A 33.611,B 20.134,C -0.7568,E1 20.2773,E2 414.4254} C_DIS
LIN {X 107.614,Y 81.5081,Z 162,A 35.3322,B 20.1339,C -0.7594,E1 20.2744,E2 412.7073} C_DIS
LIN {X 105.2223,Y 84.5732,Z 162,A 36.9485,B 20.1338,C -0.7618,E1 20.2716,E2 411.0937} C_DIS
LIN {X 102.7084,Y 87.609,Z 162,A 38.6903,B 20.1335,C -0.7688,E1 20.2685,E2 409.3419} C_DIS
LIN {X 99.823,Y 90.8829,Z 162,A 40.5353,B 20.1334,C -0.7726,E1 20.2651,E2 407.4961} C_DIS
LIN {X 97.1479,Y 93.737,Z 162,A 42.193,B 20.1333,C -0.7761,E1 20.2619,E2 405.8375} C_DIS
LIN {X 94.2145,Y 96.6856,Z 162,A 43.8604,B 20.1333,C -0.7755,E1 20.2586,E2 404.181} C_DIS
LIN {X 91.5198,Y 99.2394,Z 162,A 45.4256,B 20.1332,C -0.7782,E1 20.2554,E2 402.6159} C_DIS
LIN {X 88.4663,Y 101.9713,Z 162,A 47.1626,B 20.1331,C -0.7816,E1 20.2517,E2 400.878} C_DIS
LIN {X 85.6024,Y 104.3867,Z 162,A 48.7396,B 20.133,C -0.784,E1 20.2484,E2 399.3016} C_DIS
LIN {X 82.8802,Y 106.5609,Z 162,A 50.3151,B 20.1327,C -0.791,E1 20.2449,E2 397.7132} C_DIS
LIN {X 79.5748,Y 109.052,Z 162,A 51.9588,B 20.1327,C -0.7891,E1 20.2412,E2 396.0827} C_DIS
LIN {X 76.7455,Y 111.0613,Z 162,A 53.4788,B 20.1326,C -0.7937,E1 20.2377,E2 394.5561} C_DIS
LIN {X 73.3209,Y 113.3507,Z 162,A 55.2423,B 20.1325,C -0.7971,E1 20.2336,E2 392.7899} C_DIS
LIN {X 69.6633,Y 115.6347,Z 162,A 57.0638,B 20.1324,C -0.7995,E1 20.2293,E2 390.9687} C_DIS
LIN {X 65.7703,Y 117.893,Z 162,A 59.0213,B 20.1322,C -0.8044,E1 20.2245,E2 389.0048} C_DIS
LIN {X 61.6404,Y 120.1017,Z 162,A 60.7141,B 20.1326,C -0.7941,E1 20.2204,E2 387.3477} C_DIS
LIN {X 58.5927,Y 121.6176,Z 162,A 62.3059,B 20.1323,C -0.8023,E1 20.2164,E2 385.7374} C_DIS
LIN {X 55.577,Y 123.0253,Z 162,A 63.5842,B 20.1324,C -0.7981,E1 20.2132,E2 384.4755} C_DIS
LIN {X 52.4029,Y 124.4101,Z 162,A 65.0151,B 20.1324,C -0.7981,E1 20.2095,E2 383.0491} C_DIS
LIN {X 49.6921,Y 125.5196,Z 162,A 66.4158,B 20.1321,C -0.8062,E1 20.2058,E2 381.6289} C_DIS
LIN {X 46.0997,Y 126.8807,Z 162,A 67.9897,B 20.1321,C -0.8053,E1 20.2017,E2 380.0618} C_DIS
LIN {X 43.0597,Y 127.9447,Z 162,A 69.402,B 20.1321,C -0.8085,E1 20.198,E2 378.6438} C_DIS
LIN {X 40.2932,Y 128.8446,Z 162,A 70.633,B 20.132,C -0.8093,E1 20.1947,E2 377.4133} C_DIS
LIN {X 36.769,Y 129.8924,Z 162,A 72.1877,B 20.132,C -0.8103,E1 20.1905,E2 375.8594} C_DIS
LIN {X 33.4984,Y 130.7737,Z 162,A 73.6504,B 20.1319,C -0.8123,E1 20.1866,E2 374.3937} C_DIS
LIN {X 28.8986,Y 131.8669,Z 162,A 75.6216,B 20.1319,C -0.8119,E1 20.1812,E2 372.4272} C_DIS
LIN {X 26.1328,Y 132.4445,Z 162,A 76.9472,B 20.1317,C -0.8179,E1 20.1776,E2 371.0863} C_DIS
LIN {X 22.9988,Y 133.0246,Z 162,A 78.2821,B 20.1317,C -0.8176,E1 20.1739,E2 369.7538} C_DIS
LIN {X 19.8755,Y 133.5269,Z 162,A 79.5067,B 20.1319,C -0.813,E1 20.1706,E2 368.544} C_DIS
LIN {X 16.2158,Y 134.0186,Z 162,A 81.103,B 20.1318,C -0.8147,E1 20.1661,E2 366.9446} C_DIS
LIN {X 12.8421,Y 134.3837,Z 162,A 82.418,B 20.132,C -0.8096,E1 20.1625,E2 365.6454} C_DIS
LIN {X 10.228,Y 134.6085,Z 162,A 83.4793,B 20.132,C -0.8075,E1 20.1596,E2 364.5909} C_DIS
LIN {X 7.5381,Y 134.7875,Z 162,A 84.8707,B 20.1317,C -0.818,E1 20.1556,E2 363.1698} C_DIS
LIN {X 4.1434,Y 134.9329,Z 162,A 86.2379,B 20.1317,C -0.8148,E1 20.1518,E2 361.8123} C_DIS
LIN {X 0.6774,Y 134.9943,Z 162,A 87.6797,B 20.1318,C -0.8134,E1 20.1478,E2 360.3748} C_DIS
LIN {X -2.9964,Y 134.9648,Z 162,A 89.2316,B 20.1318,C -0.8128,E1 20.1435,E2 358.8247} C_DIS
LIN {X -6.3819,Y 134.8456,Z 162,A 90.6734,B 20.1318,C -0.8126,E1 20.1395,E2 357.3831} C_DIS
LIN {X -9.6282,Y 134.6523,Z 162,A 92.0737,B 20.1318,C -0.8129,E1 20.1356,E2 355.9812} C_DIS
LIN {X -12.906,Y 134.3775,Z 162,A 93.4688,B 20.1318,C -0.8123,E1 20.1317,E2 354.5871} C_DIS
LIN {X -17.137,Y 133.9043,Z 162,A 95.271,B 20.1319,C -0.8112,E1 20.1267,E2 352.7867} C_DIS
LIN {X -19.8755,Y 133.5269,Z 162,A 96.5824,B 20.1317,C -0.8162,E1 20.123,E2 351.4592} C_DIS
LIN {X -23.3735,Y 132.9575,Z 162,A 97.9573,B 20.132,C -0.8098,E1 20.1193,E2 350.1013} C_DIS
LIN {X -26.1328,Y 132.4445,Z 162,A 99.1523,B 20.132,C -0.8091,E1 20.116,E2 348.9068} C_DIS
LIN {X -29.6511,Y 131.6997,Z 162,A 100.6844,B 20.132,C -0.8081,E1 20.1118,E2 347.3752} C_DIS
LIN {X -32.8772,Y 130.9314,Z 162,A 102.109,B 20.132,C -0.8075,E1 20.108,E2 345.9496} C_DIS
LIN {X -35.5712,Y 130.2274,Z 162,A 103.404,B 20.132,C -0.811,E1 20.1044,E2 344.6419} C_DIS
LIN {X -39.0964,Y 129.2109,Z 162,A 104.6975,B 20.1324,C -0.7986,E1 20.1011,E2 343.3819} C_DIS
LIN {X -41.9303,Y 128.3208,Z 162,A 106.213,B 20.1321,C -0.8077,E1 20.097,E2 341.8366} C_DIS
LIN {X -45.0037,Y 127.2759,Z 162,A 107.6193,B 20.1321,C -0.8072,E1 20.0932,E2 340.4282} C_DIS
LIN {X -48.6449,Y 125.9267,Z 162,A 109.1107,B 20.1324,C -0.7987,E1 20.0894,E2 338.9575} C_DIS
LIN {X -51.6195,Y 124.7373,Z 162,A 110.5186,B 20.1324,C -0.7989,E1 20.0857,E2 337.5451} C_DIS
LIN {X -54.7168,Y 123.41,Z 162,A 111.9582,B 20.1324,C -0.7973,E1 20.0821,E2 336.1059} C_DIS
LIN {X -57.921,Y 121.9385,Z 162,A 113.4197,B 20.1326,C -0.7937,E1 20.0784,E2 334.6504} C_DIS
LIN {X -60.4848,Y 120.69,Z 162,A 114.6753,B 20.1326,C -0.7937,E1 20.0752,E2 333.3907} C_DIS
LIN {X -63.9576,Y 118.8853,Z 162,A 116.3957,B 20.1326,C -0.7934,E1 20.071,E2 331.665} C_DIS
LIN {X -67.8288,Y 116.7202,Z 162,A 118.3153,B 20.1326,C -0.7917,E1 20.0663,E2 329.7431} C_DIS
LIN {X -71.5152,Y 114.4986,Z 162,A 120.152,B 20.1328,C -0.7888,E1 20.0619,E2 327.9074} C_DIS
LIN {X -74.7667,Y 112.4023,Z 162,A 121.7245,B 20.133,C -0.783,E1 20.0583,E2 326.3455} C_DIS
LIN {X -77.6267,Y 110.4466,Z 162,A 123.2031,B 20.133,C -0.7805,E1 20.0549,E2 324.8678} C_DIS
LIN {X -80.8051,Y 108.1428,Z 162,A 124.9046,B 20.1332,C -0.7786,E1 20.0511,E2 323.1642} C_DIS
LIN {X -83.7295,Y 105.8955,Z 162,A 126.4529,B 20.1333,C -0.7747,E1 20.0477,E2 321.62} C_DIS
LIN {X -86.5952,Y 103.5645,Z 162,A 128.1163,B 20.1333,C -0.7752,E1 20.0441,E2 319.9472} C_DIS
LIN {X -89.7406,Y 100.8519,Z 162,A 129.9154,B 20.1333,C -0.7728,E1 20.0403,E2 318.1461} C_DIS
LIN {X -92.9552,Y 97.8969,Z 162,A 131.6676,B 20.1337,C -0.7645,E1 20.0367,E2 316.4088} C_DIS
LIN {X -95.4581,Y 95.4581,Z 162,A 133.1599,B 20.1337,C -0.7614,E1 20.0338,E2 314.9176} C_DIS
LIN {X -97.8969,Y 92.9552,Z 162,A 134.7053,B 20.1338,C -0.7604,E1 20.0308,E2 313.3668} C_DIS
LIN {X -100.7626,Y 89.8403,Z 162,A 136.5284,B 20.1339,C -0.7571,E1 20.0274,E2 311.543} C_DIS
LIN {X -103.5645,Y 86.5952,Z 162,A 138.317,B 20.1342,C -0.7513,E1 20.0241,E2 309.761} C_DIS
LIN {X -106.0242,Y 83.5656,Z 162,A 139.9576,B 20.1343,C -0.7464,E1 20.0213,E2 308.1248} C_DIS
LIN {X -108.1428,Y 80.8051,Z 162,A 141.5549,B 20.1343,C -0.7473,E1 20.0186,E2 306.5151} C_DIS
LIN {X -110.5662,Y 77.4571,Z 162,A 143.2095,B 20.1346,C -0.7387,E1 20.0159,E2 304.8755} C_DIS
LIN {X -112.5173,Y 74.5945,Z 162,A 144.7421,B 20.1346,C -0.7372,E1 20.0135,E2 303.3375} C_DIS
LIN {X -114.4986,Y 71.5152,Z 162,A 146.339,B 20.1347,C -0.7346,E1 20.0111,E2 301.7379} C_DIS
LIN {X -116.7202,Y 67.8288,Z 162,A 148.2059,B 20.1349,C -0.7311,E1 20.0085,E2 299.8689} C_DIS
LIN {X -119.0258,Y 63.6963,Z 162,A 150.2632,B 20.1349,C -0.7273,E1 20.0057,E2 297.8089} C_DIS
LIN {X -120.69,Y 60.4848,Z 162,A 151.7844,B 20.1352,C -0.7223,E1 20.0038,E2 296.2919} C_DIS
LIN {X -122.3444,Y 57.0597,Z 162,A 153.3019,B 20.1355,C -0.7138,E1 20.002,E2 294.7888} C_DIS
LIN {X -123.5752,Y 54.3476,Z 162,A 154.697,B 20.1355,C -0.7152,E1 20.0004,E2 293.3799} C_DIS
LIN {X -124.8924,Y 51.2481,Z 162,A 155.9962,B 20.1357,C -0.7059,E1 19.999,E2 292.0988} C_DIS
LIN {X -126.1259,Y 48.1324,Z 162,A 157.5501,B 20.1357,C -0.7068,E1 19.9975,E2 290.5312} C_DIS
LIN {X -127.4462,Y 44.5125,Z 162,A 159.0559,B 20.136,C -0.6968,E1 19.9961,E2 289.0438} C_DIS
LIN {X -128.4626,Y 41.489,Z 162,A 160.2866,B 20.1363,C -0.6878,E1 19.995,E2 287.8304} C_DIS
LIN {X -129.3261,Y 38.72,Z 162,A 161.7966,B 20.1361,C -0.6949,E1 19.9938,E2 286.2884} C_DIS
LIN {X -130.3279,Y 35.1943,Z 162,A 163.2954,B 20.1363,C -0.6879,E1 19.9926,E2 284.799} C_DIS
LIN {X -131.047,Y 32.4218,Z 162,A 164.4661,B 20.1365,C -0.6824,E1 19.9919,E2 283.6359} C_DIS
LIN {X -131.8669,Y 28.8986,Z 162,A 166.0106,B 20.1366,C -0.678,E1 19.9909,E2 282.0927} C_DIS
LIN {X -132.5509,Y 25.5765,Z 162,A 167.2449,B 20.137,C -0.6655,E1 19.9902,E2 280.8857} C_DIS
LIN {X -133.0246,Y 22.9988,Z 162,A 168.6959,B 20.1367,C -0.6752,E1 19.9895,E2 279.3953} C_DIS
LIN {X -133.6005,Y 19.361,Z 162,A 170.1418,B 20.137,C -0.6657,E1 19.9889,E2 277.9662} C_DIS
LIN {X -134.0117,Y 16.2729,Z 162,A 171.449,B 20.1372,C -0.661,E1 19.9885,E2 276.663} C_DIS
LIN {X -134.3041,Y 13.6708,Z 162,A 172.6027,B 20.1372,C -0.6591,E1 19.9881,E2 275.506} C_DIS
LIN {X -134.6085,Y 10.228,Z 162,A 173.9388,B 20.1376,C -0.6494,E1 19.9878,E2 274.1881} C_DIS
LIN {X -134.7954,Y 7.3795,Z 162,A 175.3595,B 20.1374,C -0.6537,E1 19.9876,E2 272.7439} C_DIS
LIN {X -134.9329,Y 4.1434,Z 162,A 176.5442,B 20.1378,C -0.6419,E1 19.9874,E2 271.5845} C_DIS
LIN {X -134.9898,Y 1.4949,Z 162,A 177.8699,B 20.1376,C -0.6462,E1 19.9874,E2 270.236} C_DIS
LIN {X -134.9838,Y -1.8542,Z 162,A 179.1101,B 20.138,C -0.6347,E1 19.9874,E2 269.0201} C_DIS
LIN {X -134.9124,Y -4.7732,Z 162,A -179.4255,B 20.1379,C -0.6396,E1 19.9875,E2 267.5301} C_DIS
LIN {X -134.7382,Y -8.3374,Z 162,A -177.9249,B 20.138,C -0.6343,E1 19.9878,E2 266.0335} C_DIS
LIN {X -134.4166,Y -12.4989,Z 162,A -176.3229,B 20.1384,C -0.6221,E1 19.9881,E2 264.4549} C_DIS
LIN {X -134.1378,Y -15.216,Z 162,A -174.895,B 20.1382,C -0.629,E1 19.9886,E2 262.9959} C_DIS
LIN {X -133.6962,Y -18.6912,Z 162,A -173.4726,B 20.1384,C -0.6219,E1 19.9891,E2 261.5837} C_DIS
LIN {X -133.2093,Y -21.8914,Z 162,A -172.1449,B 20.1386,C -0.6158,E1 19.9897,E2 260.2635} C_DIS
LIN {X -132.6726,Y -24.9399,Z 162,A -170.9412,B 20.1388,C -0.6074,E1 19.9903,E2 259.0753} C_DIS
LIN {X -132.1251,Y -27.7029,Z 162,A -169.4691,B 20.1386,C -0.6147,E1 19.9911,E2 257.5711} C_DIS
LIN {X -131.3356,Y -31.2244,Z 162,A -168.19,B 20.139,C -0.6001,E1 19.9919,E2 256.325} C_DIS
LIN {X -130.6474,Y -33.9964,Z 162,A -166.8183,B 20.139,C -0.6027,E1 19.9928,E2 254.9356} C_DIS
LIN {X -129.6767,Y -37.5225,Z 162,A -165.2517,B 20.139,C -0.5986,E1 19.994,E2 253.3691} C_DIS
LIN {X -128.8446,Y -40.2932,Z 162,A -164.0128,B 20.1392,C -0.5954,E1 19.995,E2 252.1306} C_DIS
LIN {X -127.6748,Y -43.853,Z 162,A -162.3812,B 20.1392,C -0.5924,E1 19.9965,E2 250.496} C_DIS
LIN {X -126.5713,Y -46.9435,Z 162,A -161.0028,B 20.1394,C -0.5878,E1 19.9978,E2 249.1212} C_DIS
LIN {X -125.3695,Y -50.0644,Z 162,A -159.5712,B 20.1394,C -0.5842,E1 19.9993,E2 247.6899} C_DIS
LIN {X -124.0841,Y -53.1704,Z 162,A -158.1323,B 20.1396,C -0.5806,E1 20.0008,E2 246.2513} C_DIS
LIN {X -122.8852,Y -55.8902,Z 162,A -156.8604,B 20.1396,C -0.5775,E1 20.0023,E2 244.9798} C_DIS
LIN {X -121.2624,Y -59.3243,Z 162,A -155.3904,B 20.1399,C -0.5674,E1 20.004,E2 243.529} C_DIS
LIN {X -119.9166,Y -62.0039,Z 162,A -153.8261,B 20.1397,C -0.5755,E1 20.0061,E2 241.9303} C_DIS
LIN {X -117.7924,Y -65.9492,Z 162,A -151.9222,B 20.1398,C -0.5705,E1 20.0086,E2 240.0284} C_DIS
LIN {X -115.4435,Y -69.9793,Z 162,A -150.002,B 20.14,C -0.5629,E1 20.0113,E2 238.1177} C_DIS
LIN {X -113.3507,Y -73.3209,Z 162,A -148.3552,B 20.1402,C -0.5575,E1 20.0138,E2 236.4759} C_DIS
LIN {X -111.1355,Y -76.6374,Z 162,A -146.6354,B 20.1402,C -0.5544,E1 20.0165,E2 234.7546} C_DIS
LIN {X -108.8182,Y -79.893,Z 162,A -144.8687,B 20.1403,C -0.5531,E1 20.0194,E2 232.9808} C_DIS
LIN {X -106.4333,Y -83.0448,Z 162,A -143.1372,B 20.1403,C -0.5512,E1 20.0224,E2 231.2441} C_DIS
LIN {X -103.6987,Y -86.4353,Z 162,A -141.3936,B 20.1406,C -0.5427,E1 20.0254,E2 229.5152} C_DIS
LIN {X -101.2917,Y -89.2432,Z 162,A -139.7279,B 20.1406,C -0.543,E1 20.0285,E2 227.8389} C_DIS
LIN {X -98.3529,Y -92.4719,Z 162,A -137.8428,B 20.1406,C -0.5403,E1 20.0321,E2 225.9513} C_DIS
LIN {X -95.4581,Y -95.4581,Z 162,A -136.053,B 20.1407,C -0.5375,E1 20.0356,E2 224.1599} C_DIS
LIN {X -92.3198,Y -98.4963,Z 162,A -134.2335,B 20.1408,C -0.5323,E1 20.0393,E2 222.346} C_DIS
LIN {X -89.0867,Y -101.43,Z 162,A -132.3966,B 20.141,C -0.528,E1 20.0431,E2 220.5123} C_DIS
LIN {X -85.9246,Y -104.1216,Z 162,A -130.5999,B 20.141,C -0.5261,E1 20.0469,E2 218.7124} C_DIS
LIN {X -82.5258,Y -106.8356,Z 162,A -128.7452,B 20.141,C -0.5232,E1 20.051,E2 216.8577} C_DIS
LIN {X -79.04,Y -109.4396,Z 162,A -126.9447,B 20.1412,C -0.5181,E1 20.0551,E2 215.064} C_DIS
LIN {X -75.6748,Y -111.7927,Z 162,A -125.1553,B 20.1412,C -0.5172,E1 20.0592,E2 213.2696} C_DIS
LIN {X -72.2455,Y -114.0392,Z 162,A -123.4754,B 20.1414,C -0.512,E1 20.0631,E2 211.5979} C_DIS
LIN {X -68.9248,Y -116.0764,Z 162,A -121.7911,B 20.1414,C -0.5108,E1 20.0671,E2 209.9104} C_DIS
LIN {X -65.5909,Y -117.9923,Z 162,A -120.0675,B 20.1414,C -0.5124,E1 20.0714,E2 208.1759} C_DIS
LIN {X -61.6404,Y -120.1017,Z 162,A -118.2394,B 20.1414,C -0.5069,E1 20.0759,E2 206.3573} C_DIS
LIN {X -58.5927,Y -121.6176,Z 162,A -116.8269,B 20.1415,C -0.5038,E1 20.0794,E2 204.9492} C_DIS
LIN {X -55.4268,Y -123.0924,Z 162,A -115.5331,B 20.1418,C -0.4942,E1 20.0826,E2 203.6792} C_DIS
LIN {X -52.8001,Y -124.2442,Z 162,A -114.1219,B 20.1416,C -0.501,E1 20.0863,E2 202.2442} C_DIS
LIN {X -49.2064,Y -125.7084,Z 162,A -112.4522,B 20.1416,C -0.5003,E1 20.0906,E2 200.5717} C_DIS
LIN {X -46.1948,Y -126.8464,Z 162,A -111.2549,B 20.1418,C -0.492,E1 20.0937,E2 199.3956} C_DIS
LIN {X -43.0597,Y -127.9447,Z 162,A -109.6935,B 20.1418,C -0.4971,E1 20.0979,E2 197.8154} C_DIS
LIN {X -39.879,Y -128.9714,Z 162,A -108.3204,B 20.1418,C -0.4941,E1 20.1015,E2 196.448} C_DIS
LIN {X -36.6942,Y -129.9133,Z 162,A -106.886,B 20.1418,C -0.4941,E1 20.1054,E2 195.0104} C_DIS
LIN {X -33.6196,Y -130.743,Z 162,A -105.6582,B 20.1419,C -0.4881,E1 20.1086,E2 193.798} C_DIS
LIN {X -30.8478,Y -131.4264,Z 162,A -104.1827,B 20.1417,C -0.4986,E1 20.1127,E2 192.2894} C_DIS
LIN {X -27.3272,Y -132.2015,Z 162,A -102.9151,B 20.1419,C -0.4868,E1 20.1161,E2 191.0543} C_DIS
LIN {X -24.5647,Y -132.7443,Z 162,A -101.5762,B 20.1419,C -0.4924,E1 20.1198,E2 189.6973} C_DIS
LIN {X -21.0623,Y -133.3432,Z 162,A -100.0006,B 20.1418,C -0.4948,E1 20.1242,E2 188.1128} C_DIS
LIN {X -17.7294,Y -133.8266,Z 162,A -98.6088,B 20.1418,C -0.4929,E1 20.128,E2 186.7252} C_DIS
LIN {X -13.6708,Y -134.3041,Z 162,A -96.9093,B 20.1418,C -0.4911,E1 20.1327,E2 185.0297} C_DIS
LIN {X -10.228,Y -134.6085,Z 162,A -95.5836,B 20.142,C -0.4849,E1 20.1364,E2 183.721} C_DIS
LIN {X -7.5381,Y -134.7875,Z 162,A -94.1652,B 20.1417,C -0.4967,E1 20.1404,E2 182.2678} C_DIS
LIN {X -3.7918,Y -134.9427,Z 162,A -92.8784,B 20.142,C -0.4837,E1 20.1439,E2 181.0185} C_DIS
LIN {X -1.4949,Y -134.9898,Z 162,A -91.6335,B 20.1417,C -0.4955,E1 20.1475,E2 179.7393} C_DIS
LIN {X 0.9393,Y -134.9913,Z 162,A -90.9282,B 20.1421,C -0.4816,E1 20.1494,E2 179.0745} C_DIS
Enddeposition()
LIN {X 0.9393,Y -134.9913,Z 162,A -90.9282,B 20.1421,C -0.4816,E1 20.1494,E2 179.0745} C_DIS
Startdeposition()
$VEL.CP = VEL_PRINT
LIN {X 0.4294,Y -134.0729,Z 162,A -91.2781,B 18.9494,C -0.3195,E1 18.9516,E2 179.8089} C_DIS
LIN {X -3.6872,Y -134.0225,Z 162,A -92.9593,B 18.9494,C -0.3224,E1 18.947,E2 181.4813} C_DIS
LIN {X -7.9214,Y -133.8393,Z 162,A -94.8016,B 18.9494,C -0.3212,E1 18.9418,E2 183.3281} C_DIS
LIN {X -11.8425,Y -133.5503,Z 162,A -96.5181,B 18.9494,C -0.3198,E1 18.937,E2 185.0498} C_DIS
LIN {X -15.828,Y -133.1355,Z 162,A -98.1526,B 18.9493,C -0.3232,E1 18.9325,E2 186.6752} C_DIS
LIN {X -19.7136,Y -132.618,Z 162,A -99.9535,B 18.9493,C -0.3186,E1 18.9275,E2 188.4921} C_DIS
LIN {X -23.5758,Y -131.9839,Z 162,A -101.392,B 18.9493,C -0.3285,E1 18.9236,E2 189.9022} C_DIS
LIN {X -26.809,Y -131.3653,Z 162,A -102.8939,B 18.9493,C -0.3253,E1 18.9195,E2 191.4161} C_DIS
LIN {X -30.198,Y -130.6283,Z 162,A -104.4192,B 18.9493,C -0.3244,E1 18.9153,E2 192.9469} C_DIS
LIN {X -35.3321,Y -129.3361,Z 162,A -106.7562,B 18.9493,C -0.3228,E1 18.9089,E2 195.2933} C_DIS
LIN {X -39.0312,Y -128.2659,Z 162,A -108.125,B 18.9491,C -0.3348,E1 18.9054,E2 196.6283} C_DIS
LIN {X -41.5448,Y -127.4761,Z 162,A -109.5883,B 18.9493,C -0.3225,E1 18.9014,E2 198.133} C_DIS
LIN {X -45.9043,Y -125.9703,Z 162,A -111.5427,B 18.9493,C -0.3249,E1 18.8962,E2 200.0851} C_DIS
LIN {X -49.8992,Y -124.4412,Z 162,A -113.0634,B 18.949,C -0.3386,E1 18.8924,E2 201.5681} C_DIS
LIN {X -52.9738,Y -123.1638,Z 162,A -114.7343,B 18.9492,C -0.3305,E1 18.888,E2 203.2692} C_DIS
LIN {X -55.8047,Y -121.9081,Z 162,A -116.0504,B 18.9492,C -0.3322,E1 18.8846,E2 204.5843} C_DIS
LIN {X -59.0781,Y -120.355,Z 162,A -117.6106,B 18.9492,C -0.3336,E1 18.8807,E2 206.1455} C_DIS
LIN {X -62.1524,Y -118.7964,Z 162,A -119.0205,B 18.949,C -0.3379,E1 18.8772,E2 207.5474} C_DIS
LIN {X -65.9316,Y -116.7438,Z 162,A -120.8382,B 18.949,C -0.3411,E1 18.8728,E2 209.3622} C_DIS
LIN {X -68.4327,Y -115.2948,Z 162,A -122.7149,B 18.9494,C -0.3186,E1 18.8681,E2 211.3162} C_DIS
LIN {X -72.6228,Y -112.7036,Z 162,A -124.3411,B 18.949,C -0.3399,E1 18.8644,E2 212.8838} C_DIS
LIN {X -76.1321,Y -110.3631,Z 162,A -126.1683,B 18.949,C -0.3419,E1 18.8602,E2 214.7131} C_DIS
LIN {X -79.8933,Y -107.6713,Z 162,A -128.1388,B 18.949,C -0.3454,E1 18.8557,E2 216.6819} C_DIS
LIN {X -83.6331,Y -104.7929,Z 162,A -130.2266,B 18.949,C -0.3464,E1 18.8511,E2 218.7773} C_DIS
LIN {X -87.2308,Y -101.818,Z 162,A -132.1417,B 18.9488,C -0.3531,E1 18.8471,E2 220.6815} C_DIS
LIN {X -90.2389,Y -99.1614,Z 162,A -133.8363,B 18.9488,C -0.3572,E1 18.8436,E2 222.3727} C_DIS
LIN {X -93.4883,Y -96.1043,Z 162,A -135.8014,B 18.9487,C -0.3589,E1 18.8396,E2 224.3435} C_DIS
LIN {X -96.6467,Y -92.9279,Z 162,A -137.7575,B 18.9487,C -0.3614,E1 18.8358,E2 226.3033} C_DIS
LIN {X -99.7165,Y -89.6252,Z 162,A -139.6949,B 18.9486,C -0.3652,E1 18.8321,E2 228.2405} C_DIS
LIN {X -102.8694,Y -85.9881,Z 162,A -141.724,B 18.9485,C -0.3709,E1 18.8284,E2 230.2645} C_DIS
LIN {X -105.4354,Y -82.8214,Z 162,A -143.4624,B 18.9484,C -0.3751,E1 18.8254,E2 232.001} C_DIS
LIN {X -108.2056,Y -79.1684,Z 162,A -145.4019,B 18.9483,C -0.3805,E1 18.8222,E2 233.9364} C_DIS
LIN {X -110.0925,Y -76.5222,Z 162,A -146.8573,B 18.9483,C -0.3815,E1 18.8198,E2 235.3985} C_DIS
LIN {X -112.3542,Y -73.1614,Z 162,A -148.7728,B 18.9483,C -0.3791,E1 18.8169,E2 237.3345} C_DIS
LIN {X -114.072,Y -70.4539,Z 162,A -150.0093,B 18.9481,C -0.3875,E1 18.8151,E2 238.5536} C_DIS
LIN {X -116.4172,Y -66.506,Z 162,A -151.9417,B 18.9481,C -0.3937,E1 18.8124,E2 240.4803} C_DIS
LIN {X -118.5271,Y -62.6653,Z 162,A -153.7692,B 18.9479,C -0.4004,E1 18.8099,E2 242.3003} C_DIS
LIN {X -119.8442,Y -60.1121,Z 162,A -155.2239,B 18.9479,C -0.3954,E1 18.8081,E2 243.7811} C_DIS
LIN {X -121.9427,Y -55.7297,Z 162,A -157.1603,B 18.9478,C -0.4062,E1 18.8058,E2 245.6982} C_DIS
LIN {X -123.5916,Y -51.9683,Z 162,A -158.847,B 18.9476,C -0.4136,E1 18.804,E2 247.3746} C_DIS
LIN {X -124.8227,Y -48.938,Z 162,A -160.2604,B 18.9476,C -0.417,E1 18.8025,E2 248.7882} C_DIS
LIN {X -126.0374,Y -45.7181,Z 162,A -161.715,B 18.9474,C -0.4218,E1 18.8011,E2 250.2392} C_DIS
LIN {X -127.0987,Y -42.6796,Z 162,A -163.1406,B 18.9474,C -0.424,E1 18.7998,E2 251.6691} C_DIS
LIN {X -127.9691,Y -40.0008,Z 162,A -164.4602,B 18.9474,C -0.4233,E1 18.7987,E2 253.0011} C_DIS
LIN {X -129.1778,Y -35.8983,Z 162,A -166.2068,B 18.9472,C -0.4316,E1 18.7973,E2 254.7356} C_DIS
LIN {X -129.9778,Y -32.8836,Z 162,A -167.8922,B 18.9474,C -0.4229,E1 18.7962,E2 256.4613} C_DIS
LIN {X -130.8617,Y -29.1762,Z 162,A -169.1337,B 18.947,C -0.4417,E1 18.7954,E2 257.6544} C_DIS
LIN {X -131.6003,Y -25.6348,Z 162,A -171.1398,B 18.9473,C -0.4299,E1 18.7943,E2 259.7134} C_DIS
LIN {X -132.2879,Y -21.8069,Z 162,A -172.4062,B 18.9468,C -0.4491,E1 18.7937,E2 260.9302} C_DIS
LIN {X -132.8398,Y -18.1581,Z 162,A -173.9365,B 18.9467,C -0.4556,E1 18.7931,E2 262.4529} C_DIS
LIN {X -133.3128,Y -14.2581,Z 162,A -175.6617,B 18.9466,C -0.4592,E1 18.7926,E2 264.1812} C_DIS
LIN {X -133.6875,Y -10.1693,Z 162,A -177.4729,B 18.9466,C -0.4626,E1 18.7921,E2 265.9966} C_DIS
LIN {X -133.9161,Y -6.4925,Z 162,A -179.0203,B 18.9464,C -0.4684,E1 18.7919,E2 267.5385} C_DIS
LIN {X -134.0481,Y -2.6284,Z 162,A 179.3715,B 18.9462,C -0.4751,E1 18.7918,E2 269.139} C_DIS
LIN {X -134.0698,Y 1.0742,Z 162,A 177.6614,B 18.9462,C -0.4755,E1 18.7918,E2 270.8621} C_DIS
LIN {X -133.9859,Y 4.8525,Z 162,A 176.1368,B 18.946,C -0.4838,E1 18.7918,E2 272.3734} C_DIS
LIN {X -133.8521,Y 7.7147,Z 162,A 174.7414,B 18.946,C -0.4815,E1 18.7921,E2 273.7874} C_DIS
LIN {X -133.5428,Y 11.9307,Z 162,A 173.0643,B 18.9458,C -0.4917,E1 18.7925,E2 275.4463} C_DIS
LIN {X -133.2963,Y 14.4117,Z 162,A 171.878,B 18.9458,C -0.4907,E1 18.7928,E2 276.6454} C_DIS
LIN {X -132.7506,Y 18.7853,Z 162,A 170.0234,B 18.9457,C -0.4976,E1 18.7935,E2 278.4937} C_DIS
LIN {X -132.2159,Y 22.2387,Z 162,A 168.174,B 18.9459,C -0.4896,E1 18.7943,E2 280.383} C_DIS
LIN {X -131.5434,Y 25.9323,Z 162,A 166.8597,B 18.9455,C -0.5048,E1 18.795,E2 281.6605} C_DIS
LIN {X -130.916,Y 28.9305,Z 162,A 165.2653,B 18.9456,C -0.4987,E1 18.796,E2 283.2868} C_DIS
LIN {X -130.1242,Y 32.3067,Z 162,A 164.136,B 18.9452,C -0.5158,E1 18.7967,E2 284.3719} C_DIS
LIN {X -129.3613,Y 35.236,Z 162,A 161.8705,B 18.946,C -0.4852,E1 18.7985,E2 286.7503} C_DIS
LIN {X -127.4787,Y 41.5369,Z 162,A 159.8239,B 18.9451,C -0.5208,E1 18.8001,E2 288.7025} C_DIS
LIN {X -126.3332,Y 44.8977,Z 162,A 158.4483,B 18.9448,C -0.5304,E1 18.8014,E2 290.0589} C_DIS
LIN {X -125.2988,Y 47.7101,Z 162,A 157.0147,B 18.9448,C -0.5287,E1 18.8028,E2 291.5087} C_DIS
LIN {X -122.6804,Y 54.088,Z 162,A 154.0578,B 18.9446,C -0.537,E1 18.806,E2 294.4623} C_DIS
LIN {X -121.3081,Y 57.1,Z 162,A 151.9819,B 18.9451,C -0.5174,E1 18.8086,E2 296.6142} C_DIS
LIN {X -118.8143,Y 62.1184,Z 162,A 150.3276,B 18.9442,C -0.5507,E1 18.8106,E2 298.1773} C_DIS
LIN {X -116.8594,Y 65.7259,Z 162,A 148.5198,B 18.9442,C -0.5536,E1 18.813,E2 299.9889} C_DIS
LIN {X -114.7934,Y 69.2711,Z 162,A 146.6146,B 18.9442,C -0.553,E1 18.8157,E2 301.9095} C_DIS
LIN {X -112.1849,Y 73.4212,Z 162,A 144.5727,B 18.944,C -0.5606,E1 18.8188,E2 303.942} C_DIS
LIN {X -109.5564,Y 77.2877,Z 162,A 142.5866,B 18.9438,C -0.5663,E1 18.822,E2 305.9237} C_DIS
LIN {X -106.8493,Y 80.9895,Z 162,A 140.6274,B 18.9437,C -0.5714,E1 18.8252,E2 307.8799} C_DIS
LIN {X -104.5997,Y 83.8753,Z 162,A 138.518,B 18.9441,C -0.5556,E1 18.829,E2 310.0515} C_DIS
LIN {X -101.484,Y 87.6186,Z 162,A 137.0088,B 18.9434,C -0.5814,E1 18.8316,E2 311.4901} C_DIS
LIN {X -97.9036,Y 91.6007,Z 162,A 134.5362,B 18.9434,C -0.5802,E1 18.8363,E2 313.9812} C_DIS
LIN {X -93.9184,Y 95.6823,Z 162,A 131.8303,B 18.9435,C -0.5761,E1 18.8417,E2 316.7154} C_DIS
LIN {X -90.9409,Y 98.5182,Z 162,A 130.7302,B 18.9427,C -0.604,E1 18.8438,E2 317.7353} C_DIS
LIN {X -85.6457,Y 103.1545,Z 162,A 126.8842,B 18.9434,C -0.5798,E1 18.8521,E2 321.6767} C_DIS
LIN {X -81.8596,Y 106.1844,Z 162,A 125.3132,B 18.9427,C -0.6023,E1 18.8555,E2 323.1859} C_DIS
LIN {X -78.4704,Y 108.7128,Z 162,A 123.5473,B 18.9426,C -0.6073,E1 18.8594,E2 324.9445} C_DIS
LIN {X -74.9577,Y 111.1639,Z 162,A 121.6495,B 18.9426,C -0.6083,E1 18.8638,E2 326.8481} C_DIS
LIN {X -71.2352,Y 113.5856,Z 162,A 119.723,B 18.9425,C -0.6106,E1 18.8683,E2 328.7758} C_DIS
LIN {X -67.5566,Y 115.8114,Z 162,A 117.9054,B 18.9424,C -0.6145,E1 18.8727,E2 330.5888} C_DIS
LIN {X -64.1355,Y 117.7397,Z 162,A 116.1509,B 18.9424,C -0.6145,E1 18.877,E2 332.3504} C_DIS
LIN {X -57.7044,Y 121.0194,Z 162,A 113.2463,B 18.942,C -0.6259,E1 18.8842,E2 335.2301} C_DIS
LIN {X -55.0278,Y 122.2601,Z 162,A 112.1269,B 18.9418,C -0.6329,E1 18.887,E2 336.3314} C_DIS
LIN {X -51.9771,Y 123.588,Z 162,A 110.3469,B 18.9421,C -0.6214,E1 18.8916,E2 338.1526} C_DIS
LIN {X -47.4479,Y 125.397,Z 162,A 108.4228,B 18.9419,C -0.6301,E1 18.8966,E2 340.0556} C_DIS
LIN {X -44.6781,Y 126.4121,Z 162,A 107.1745,B 18.9418,C -0.632,E1 18.8999,E2 341.3012} C_DIS
LIN {X -40.0457,Y 127.9548,Z 162,A 104.9791,B 18.9418,C -0.6302,E1 18.9057,E2 343.5077} C_DIS
LIN {X -36.3394,Y 129.0544,Z 162,A 103.3472,B 18.9418,C -0.6326,E1 18.9101,E2 345.1357} C_DIS
LIN {X -32.5308,Y 130.0673,Z 162,A 101.7248,B 18.9417,C -0.6365,E1 18.9145,E2 346.7493} C_DIS
LIN {X -28.9139,Y 130.9196,Z 162,A 99.9247,B 18.9419,C -0.6297,E1 18.9194,E2 348.5734} C_DIS
LIN {X -23.9906,Y 131.9097,Z 162,A 97.8719,B 18.9417,C -0.6348,E1 18.925,E2 350.6134} C_DIS
LIN {X -19.6723,Y 132.6239,Z 162,A 95.9933,B 18.9417,C -0.6356,E1 18.9302,E2 352.4918} C_DIS
LIN {X -15.4577,Y 133.1797,Z 162,A 94.1628,B 18.9417,C -0.6361,E1 18.9353,E2 354.3227} C_DIS
LIN {X -11.3553,Y 133.5914,Z 162,A 92.4954,B 18.9415,C -0.6405,E1 18.9399,E2 355.9776} C_DIS
LIN {X -7.4458,Y 133.8682,Z 162,A 90.8061,B 18.9415,C -0.6405,E1 18.9446,E2 357.6678} C_DIS
LIN {X -3.8029,Y 134.0193,Z 162,A 89.2414,B 18.9415,C -0.6405,E1 18.9489,E2 359.2323} C_DIS
LIN {X 0.4858,Y 134.0726,Z 162,A 87.4198,B 18.9415,C -0.6413,E1 18.954,E2 361.0517} C_DIS
LIN {X 4.3571,Y 134.0039,Z 162,A 85.6832,B 18.9415,C -0.6382,E1 18.9589,E2 362.7974} C_DIS
LIN {X 7.6995,Y 133.853,Z 162,A 84.2195,B 18.9416,C -0.6368,E1 18.963,E2 364.2645} C_DIS
LIN {X 12.3157,Y 133.5072,Z 162,A 82.3342,B 18.9416,C -0.6402,E1 18.9682,E2 366.138} C_DIS
LIN {X 15.8615,Y 133.1315,Z 162,A 80.8674,B 18.9415,C -0.6421,E1 18.9723,E2 367.5975} C_DIS
LIN {X 19.1958,Y 132.6919,Z 162,A 79.4039,B 18.9415,C -0.6407,E1 18.9763,E2 369.0637} C_DIS
LIN {X 23.324,Y 132.029,Z 162,A 77.6224,B 18.9415,C -0.6402,E1 18.9812,E2 370.8442} C_DIS
LIN {X 26.5756,Y 131.4128,Z 162,A 76.2424,B 18.9415,C -0.6409,E1 18.985,E2 372.2198} C_DIS
LIN {X 29.2505,Y 130.8447,Z 162,A 74.8068,B 18.9419,C -0.6297,E1 18.989,E2 373.6872} C_DIS
LIN {X 34.3226,Y 129.6053,Z 162,A 72.8329,B 18.9416,C -0.6385,E1 18.9942,E2 375.63} C_DIS
LIN {X 37.1951,Y 128.8111,Z 162,A 71.4771,B 18.9417,C -0.6343,E1 18.9979,E2 376.9956} C_DIS
LIN {X 40.6077,Y 127.7755,Z 162,A 69.9482,B 18.9417,C -0.6329,E1 19.002,E2 378.525} C_DIS
LIN {X 45.0487,Y 126.2787,Z 162,A 67.9983,B 18.9417,C -0.6332,E1 19.0071,E2 380.4687} C_DIS
LIN {X 48.4203,Y 125.024,Z 162,A 66.471,B 18.9417,C -0.6321,E1 19.0111,E2 381.9949} C_DIS
LIN {X 52.1722,Y 123.5065,Z 162,A 64.649,B 18.942,C -0.6266,E1 19.0158,E2 383.8282} C_DIS
LIN {X 56.0976,Y 121.7726,Z 162,A 62.8974,B 18.942,C -0.6278,E1 19.0203,E2 385.5702} C_DIS
LIN {X 59.9102,Y 119.9445,Z 162,A 61.18,B 18.9419,C -0.6291,E1 19.0246,E2 387.2772} C_DIS
LIN {X 63.4621,Y 118.1041,Z 162,A 59.5565,B 18.9419,C -0.6303,E1 19.0285,E2 388.8908} C_DIS
LIN {X 69.9057,Y 114.4083,Z 162,A 56.18,B 18.9423,C -0.6175,E1 19.0368,E2 392.2929} C_DIS
LIN {X 73.7707,Y 111.9549,Z 162,A 54.2724,B 18.9423,C -0.6164,E1 19.0412,E2 394.1953} C_DIS
LIN {X 77.5415,Y 109.3774,Z 162,A 52.2989,B 18.9424,C -0.6122,E1 19.0458,E2 396.1724} C_DIS
LIN {X 81.1358,Y 106.7387,Z 162,A 50.3974,B 18.9425,C -0.6091,E1 19.05,E2 398.0743} C_DIS
LIN {X 84.5688,Y 104.0396,Z 162,A 48.5409,B 18.9426,C -0.606,E1 19.0541,E2 399.9306} C_DIS
LIN {X 87.5863,Y 101.5118,Z 162,A 46.874,B 18.9426,C -0.6034,E1 19.0576,E2 401.5967} C_DIS
LIN {X 90.9749,Y 98.4869,Z 162,A 44.9421,B 18.9428,C -0.5999,E1 19.0616,E2 403.5287} C_DIS
LIN {X 94.213,Y 95.3944,Z 162,A 43.0086,B 18.9429,C -0.5951,E1 19.0655,E2 405.4659} C_DIS
LIN {X 97.4054,Y 92.1316,Z 162,A 41.1064,B 18.943,C -0.593,E1 19.0692,E2 407.3637} C_DIS
LIN {X 100.4099,Y 88.8474,Z 162,A 39.2331,B 18.9431,C -0.5899,E1 19.0726,E2 409.2349} C_DIS
LIN {X 103.2902,Y 85.4819,Z 162,A 37.3694,B 18.9431,C -0.5868,E1 19.076,E2 411.0966} C_DIS
LIN {X 106.0669,Y 82.0112,Z 162,A 35.4609,B 18.9433,C -0.5819,E1 19.0793,E2 413.0078} C_DIS
LIN {X 108.7641,Y 78.3996,Z 162,A 33.5923,B 18.9434,C -0.5797,E1 19.0824,E2 414.8712} C_DIS
LIN {X 111.2088,Y 74.8913,Z 162,A 31.7066,B 18.9436,C -0.5727,E1 19.0854,E2 416.7657} C_DIS
LIN {X 113.6308,Y 71.1632,Z 162,A 29.8526,B 18.9436,C -0.5697,E1 19.0882,E2 418.616} C_DIS
LIN {X 115.7633,Y 67.6385,Z 162,A 27.9699,B 18.944,C -0.56,E1 19.0909,E2 420.5154} C_DIS
LIN {X 117.9145,Y 63.8149,Z 162,A 26.383,B 18.9438,C -0.5671,E1 19.093,E2 422.0692} C_DIS
LIN {X 121.4551,Y 56.7843,Z 162,A 22.9611,B 18.9441,C -0.5555,E1 19.0972,E2 425.502} C_DIS
LIN {X 122.7663,Y 53.8932,Z 162,A 21.6739,B 18.9441,C -0.5546,E1 19.0987,E2 426.7824} C_DIS
LIN {X 124.2335,Y 50.4146,Z 162,A 19.9869,B 18.9443,C -0.547,E1 19.1005,E2 428.4803} C_DIS
LIN {X 125.5335,Y 47.0834,Z 162,A 18.5456,B 18.9443,C -0.5463,E1 19.1019,E2 429.9128} C_DIS
LIN {X 127.5356,Y 41.3587,Z 162,A 15.8139,B 18.9447,C -0.5328,E1 19.1044,E2 432.6649} C_DIS
LIN {X 128.6941,Y 37.5945,Z 162,A 14.1984,B 18.9447,C -0.5307,E1 19.1057,E2 434.2742} C_DIS
LIN {X 129.8901,Y 33.2288,Z 162,A 12.5657,B 18.9446,C -0.5378,E1 19.1069,E2 435.8725} C_DIS
LIN {X 130.666,Y 30.033,Z 162,A 10.564,B 18.9454,C -0.5082,E1 19.1082,E2 437.949} C_DIS
LIN {X 131.4802,Y 26.2443,Z 162,A 9.1856,B 18.9452,C -0.5149,E1 19.1089,E2 439.2958} C_DIS
LIN {X 132.1605,Y 22.5705,Z 162,A 7.7379,B 18.9452,C -0.5164,E1 19.1096,E2 440.7275} C_DIS
LIN {X 132.7066,Y 19.093,Z 162,A 6.2268,B 18.9452,C -0.5115,E1 19.1103,E2 442.2415} C_DIS
LIN {X 133.1784,Y 15.4687,Z 162,A 4.6154,B 18.9455,C -0.5046,E1 19.1108,E2 443.8613} C_DIS
LIN {X 133.5884,Y 11.3908,Z 162,A 2.9938,B 18.9455,C -0.5047,E1 19.1112,E2 445.4694} C_DIS
LIN {X 133.8242,Y 8.1669,Z 162,A 1.5147,B 18.9457,C -0.4962,E1 19.1115,E2 446.9625} C_DIS
LIN {X 134.0186,Y 3.8279,Z 162,A -0.2925,B 18.9457,C -0.4926,E1 19.1117,E2 448.7664} C_DIS
LIN {X 134.0744,Y -0.3915,Z 162,A -2.1296,B 18.946,C -0.4855,E1 19.1117,E2 450.6104} C_DIS
LIN {X 134.0122,Y -4.0588,Z 162,A -3.7203,B 18.9461,C -0.4796,E1 19.1117,E2 452.2063} C_DIS
LIN {X 133.8263,Y -8.1327,Z 162,A -5.3417,B 18.9461,C -0.4793,E1 19.1114,E2 453.8153} C_DIS
LIN {X 133.5353,Y -12.0201,Z 162,A -6.9895,B 18.9462,C -0.4749,E1 19.111,E2 455.4635} C_DIS
LIN {X 133.1252,Y -15.9143,Z 162,A -8.6035,B 18.9462,C -0.4722,E1 19.1105,E2 457.0728} C_DIS
LIN {X 132.7629,Y -18.699,Z 162,A -9.808,B 18.9464,C -0.4683,E1 19.1101,E2 458.2796} C_DIS
LIN {X 132.1149,Y -22.844,Z 162,A -11.7249,B 18.9466,C -0.4573,E1 19.1092,E2 460.2147} C_DIS
LIN {X 131.5558,Y -25.8674,Z 162,A -12.8594,B 18.9466,C -0.4609,E1 19.1086,E2 461.3292} C_DIS
LIN {X 130.941,Y -28.8146,Z 162,A -14.3183,B 18.9468,C -0.4496,E1 19.1077,E2 462.8112} C_DIS
LIN {X 129.9641,Y -32.9374,Z 162,A -15.9681,B 18.9468,C -0.4509,E1 19.1066,E2 464.444} C_DIS
LIN {X 129.1499,Y -35.998,Z 162,A -17.188,B 18.9468,C -0.4525,E1 19.1058,E2 465.6496} C_DIS
LIN {X 128.182,Y -39.3052,Z 162,A -18.8298,B 18.947,C -0.4408,E1 19.1044,E2 467.3145} C_DIS
LIN {X 126.8205,Y -43.5,Z 162,A -20.6756,B 18.9471,C -0.4367,E1 19.1028,E2 469.1585} C_DIS
LIN {X 125.3966,Y -47.4488,Z 162,A -22.5182,B 18.9473,C -0.4293,E1 19.101,E2 471.01} C_DIS
LIN {X 124.0692,Y -50.8219,Z 162,A -24.1272,B 18.9474,C -0.4221,E1 19.0993,E2 472.6288} C_DIS
LIN {X 122.4847,Y -54.5255,Z 162,A -25.5762,B 18.9473,C -0.4287,E1 19.0978,E2 474.0468} C_DIS
LIN {X 120.7889,Y -58.1868,Z 162,A -27.4665,B 18.9475,C -0.4166,E1 19.0955,E2 475.9603} C_DIS
LIN {X 119.0947,Y -61.5843,Z 162,A -29.1146,B 18.9477,C -0.4109,E1 19.0934,E2 477.6142} C_DIS
LIN {X 117.6227,Y -64.3502,Z 162,A -30.5096,B 18.9477,C -0.4047,E1 19.0915,E2 479.0182} C_DIS
LIN {X 115.1534,Y -68.671,Z 162,A -32.4771,B 18.9477,C -0.4055,E1 19.0888,E2 480.9693} C_DIS
LIN {X 113.5333,Y -71.3182,Z 162,A -34.1685,B 18.9482,C -0.3864,E1 19.0862,E2 482.7077} C_DIS
LIN {X 111.3914,Y -74.6191,Z 162,A -35.4995,B 18.948,C -0.3967,E1 19.0842,E2 483.9981} C_DIS
LIN {X 108.9205,Y -78.1818,Z 162,A -37.3561,B 18.948,C -0.3916,E1 19.0812,E2 485.858} C_DIS
LIN {X 106.3979,Y -81.5814,Z 162,A -39.0908,B 18.948,C -0.3901,E1 19.0783,E2 487.5863} C_DIS
LIN {X 104.3494,Y -84.1855,Z 162,A -40.7799,B 18.9484,C -0.3749,E1 19.0753,E2 489.3111} C_DIS
LIN {X 102.1701,Y -86.8175,Z 162,A -42.0896,B 18.9484,C -0.3776,E1 19.0729,E2 490.6043} C_DIS
LIN {X 99.0538,Y -90.3575,Z 162,A -43.9343,B 18.9483,C -0.3799,E1 19.0695,E2 492.431} C_DIS
LIN {X 96.4421,Y -93.1394,Z 162,A -45.5584,B 18.9483,C -0.3763,E1 19.0664,E2 494.0565} C_DIS
LIN {X 94.1747,Y -95.4322,Z 162,A -46.9099,B 18.9483,C -0.3742,E1 19.0637,E2 495.4067} C_DIS
LIN {X 91.2236,Y -98.2563,Z 162,A -48.7019,B 18.9485,C -0.3682,E1 19.0601,E2 497.2068} C_DIS
LIN {X 87.9723,Y -101.1778,Z 162,A -50.6046,B 18.9486,C -0.3627,E1 19.0561,E2 499.1163} C_DIS
LIN {X 84.6739,Y -103.9537,Z 162,A -52.3498,B 18.9486,C -0.3628,E1 19.0524,E2 500.8521} C_DIS
LIN {X 82.1162,Y -105.9855,Z 162,A -53.9194,B 18.9488,C -0.3527,E1 19.0489,E2 502.4448} C_DIS
LIN {X 78.1581,Y -108.9375,Z 162,A -55.87,B 18.9488,C -0.3551,E1 19.0445,E2 504.3785} C_DIS
LIN {X 74.6835,Y -111.3484,Z 162,A -57.7274,B 18.9488,C -0.3496,E1 19.0402,E2 506.2444} C_DIS
LIN {X 72.239,Y -112.9493,Z 162,A -59.1423,B 18.949,C -0.3404,E1 19.0368,E2 507.6812} C_DIS
LIN {X 69.4711,Y -114.6725,Z 162,A -60.3179,B 18.9489,C -0.3469,E1 19.0341,E2 508.8317} C_DIS
LIN {X 66.7819,Y -116.2598,Z 162,A -61.7354,B 18.9489,C -0.3411,E1 19.0306,E2 510.2611} C_DIS
LIN {X 62.6945,Y -118.5118,Z 162,A -63.469,B 18.9489,C -0.3487,E1 19.0264,E2 511.9648} C_DIS
LIN {X 59.4739,Y -120.1597,Z 162,A -64.8824,B 18.9489,C -0.3518,E1 19.023,E2 513.3635} C_DIS
LIN {X 55.8954,Y -121.8661,Z 162,A -66.8026,B 18.949,C -0.3399,E1 19.018,E2 515.3135} C_DIS
LIN {X 52.0496,Y -123.5577,Z 162,A -68.6598,B 18.9491,C -0.3348,E1 19.0132,E2 517.1802} C_DIS
LIN {X 48.8112,Y -124.8721,Z 162,A -70.0525,B 18.9491,C -0.337,E1 19.0097,E2 518.5619} C_DIS
LIN {X 45.6893,Y -126.0478,Z 162,A -71.4609,B 18.9491,C -0.3359,E1 19.006,E2 519.9696} C_DIS
LIN {X 41.6067,Y -127.456,Z 162,A -73.6172,B 18.9493,C -0.321,E1 19.0002,E2 522.166} C_DIS
Enddeposition()
END
